   // UNICODE_TO_GBK[12326] := 16#6346;
   // UNICODE_TO_GBK[12327] := 16#C0A6;
   // UNICODE_TO_GBK[12328] := 16#6347;
   // UNICODE_TO_GBK[12329] := 16#92BB;
   // UNICODE_TO_GBK[12330] := 16#6348;
   // UNICODE_TO_GBK[12331] := 16#92BC;
   // UNICODE_TO_GBK[12332] := 16#6349;
   // UNICODE_TO_GBK[12333] := 16#D7BD;
   // UNICODE_TO_GBK[12334] := 16#634A;
   // UNICODE_TO_GBK[12335] := 16#92BD;
   // UNICODE_TO_GBK[12336] := 16#634B;
   // UNICODE_TO_GBK[12337] := 16#DEDB;
   // UNICODE_TO_GBK[12338] := 16#634C;
   // UNICODE_TO_GBK[12339] := 16#B0C6;
   // UNICODE_TO_GBK[12340] := 16#634D;
   // UNICODE_TO_GBK[12341] := 16#BAB4;
   // UNICODE_TO_GBK[12342] := 16#634E;
   // UNICODE_TO_GBK[12343] := 16#C9D3;
   // UNICODE_TO_GBK[12344] := 16#634F;
   // UNICODE_TO_GBK[12345] := 16#C4F3;
   // UNICODE_TO_GBK[12346] := 16#6350;
   // UNICODE_TO_GBK[12347] := 16#BEE8;
   // UNICODE_TO_GBK[12348] := 16#6351;
   // UNICODE_TO_GBK[12349] := 16#92BE;
   // UNICODE_TO_GBK[12350] := 16#6352;
   // UNICODE_TO_GBK[12351] := 16#92BF;
   // UNICODE_TO_GBK[12352] := 16#6353;
   // UNICODE_TO_GBK[12353] := 16#92C0;
   // UNICODE_TO_GBK[12354] := 16#6354;
   // UNICODE_TO_GBK[12355] := 16#92C1;
   // UNICODE_TO_GBK[12356] := 16#6355;
   // UNICODE_TO_GBK[12357] := 16#B2B6;
   // UNICODE_TO_GBK[12358] := 16#6356;
   // UNICODE_TO_GBK[12359] := 16#92C2;
   // UNICODE_TO_GBK[12360] := 16#6357;
   // UNICODE_TO_GBK[12361] := 16#92C3;
   // UNICODE_TO_GBK[12362] := 16#6358;
   // UNICODE_TO_GBK[12363] := 16#92C4;
   // UNICODE_TO_GBK[12364] := 16#6359;
   // UNICODE_TO_GBK[12365] := 16#92C5;
   // UNICODE_TO_GBK[12366] := 16#635A;
   // UNICODE_TO_GBK[12367] := 16#92C6;
   // UNICODE_TO_GBK[12368] := 16#635B;
   // UNICODE_TO_GBK[12369] := 16#92C7;
   // UNICODE_TO_GBK[12370] := 16#635C;
   // UNICODE_TO_GBK[12371] := 16#92C8;
   // UNICODE_TO_GBK[12372] := 16#635D;
   // UNICODE_TO_GBK[12373] := 16#92C9;
   // UNICODE_TO_GBK[12374] := 16#635E;
   // UNICODE_TO_GBK[12375] := 16#C0CC;
   // UNICODE_TO_GBK[12376] := 16#635F;
   // UNICODE_TO_GBK[12377] := 16#CBF0;
   // UNICODE_TO_GBK[12378] := 16#6360;
   // UNICODE_TO_GBK[12379] := 16#92CA;
   // UNICODE_TO_GBK[12380] := 16#6361;
   // UNICODE_TO_GBK[12381] := 16#BCF1;
   // UNICODE_TO_GBK[12382] := 16#6362;
   // UNICODE_TO_GBK[12383] := 16#BBBB;
   // UNICODE_TO_GBK[12384] := 16#6363;
   // UNICODE_TO_GBK[12385] := 16#B5B7;
   // UNICODE_TO_GBK[12386] := 16#6364;
   // UNICODE_TO_GBK[12387] := 16#92CB;
   // UNICODE_TO_GBK[12388] := 16#6365;
   // UNICODE_TO_GBK[12389] := 16#92CC;
   // UNICODE_TO_GBK[12390] := 16#6366;
   // UNICODE_TO_GBK[12391] := 16#92CD;
   // UNICODE_TO_GBK[12392] := 16#6367;
   // UNICODE_TO_GBK[12393] := 16#C5F5;
   // UNICODE_TO_GBK[12394] := 16#6368;
   // UNICODE_TO_GBK[12395] := 16#92CE;
   // UNICODE_TO_GBK[12396] := 16#6369;
   // UNICODE_TO_GBK[12397] := 16#DEE6;
   // UNICODE_TO_GBK[12398] := 16#636A;
   // UNICODE_TO_GBK[12399] := 16#92CF;
   // UNICODE_TO_GBK[12400] := 16#636B;
   // UNICODE_TO_GBK[12401] := 16#92D0;
   // UNICODE_TO_GBK[12402] := 16#636C;
   // UNICODE_TO_GBK[12403] := 16#92D1;
   // UNICODE_TO_GBK[12404] := 16#636D;
   // UNICODE_TO_GBK[12405] := 16#DEE3;
   // UNICODE_TO_GBK[12406] := 16#636E;
   // UNICODE_TO_GBK[12407] := 16#BEDD;
   // UNICODE_TO_GBK[12408] := 16#636F;
   // UNICODE_TO_GBK[12409] := 16#92D2;
   // UNICODE_TO_GBK[12410] := 16#6370;
   // UNICODE_TO_GBK[12411] := 16#92D3;
   // UNICODE_TO_GBK[12412] := 16#6371;
   // UNICODE_TO_GBK[12413] := 16#DEDF;
   // UNICODE_TO_GBK[12414] := 16#6372;
   // UNICODE_TO_GBK[12415] := 16#92D4;
   // UNICODE_TO_GBK[12416] := 16#6373;
   // UNICODE_TO_GBK[12417] := 16#92D5;
   // UNICODE_TO_GBK[12418] := 16#6374;
   // UNICODE_TO_GBK[12419] := 16#92D6;
   // UNICODE_TO_GBK[12420] := 16#6375;
   // UNICODE_TO_GBK[12421] := 16#92D7;
   // UNICODE_TO_GBK[12422] := 16#6376;
   // UNICODE_TO_GBK[12423] := 16#B4B7;
   // UNICODE_TO_GBK[12424] := 16#6377;
   // UNICODE_TO_GBK[12425] := 16#BDDD;
   // UNICODE_TO_GBK[12426] := 16#6378;
   // UNICODE_TO_GBK[12427] := 16#92D8;
   // UNICODE_TO_GBK[12428] := 16#6379;
   // UNICODE_TO_GBK[12429] := 16#92D9;
   // UNICODE_TO_GBK[12430] := 16#637A;
   // UNICODE_TO_GBK[12431] := 16#DEE0;
   // UNICODE_TO_GBK[12432] := 16#637B;
   // UNICODE_TO_GBK[12433] := 16#C4ED;
   // UNICODE_TO_GBK[12434] := 16#637C;
   // UNICODE_TO_GBK[12435] := 16#92DA;
   // UNICODE_TO_GBK[12436] := 16#637D;
   // UNICODE_TO_GBK[12437] := 16#92DB;
   // UNICODE_TO_GBK[12438] := 16#637E;
   // UNICODE_TO_GBK[12439] := 16#92DC;
   // UNICODE_TO_GBK[12440] := 16#637F;
   // UNICODE_TO_GBK[12441] := 16#92DD;
   // UNICODE_TO_GBK[12442] := 16#6380;
   // UNICODE_TO_GBK[12443] := 16#CFC6;
   // UNICODE_TO_GBK[12444] := 16#6381;
   // UNICODE_TO_GBK[12445] := 16#92DE;
   // UNICODE_TO_GBK[12446] := 16#6382;
   // UNICODE_TO_GBK[12447] := 16#B5E0;
   // UNICODE_TO_GBK[12448] := 16#6383;
   // UNICODE_TO_GBK[12449] := 16#92DF;
   // UNICODE_TO_GBK[12450] := 16#6384;
   // UNICODE_TO_GBK[12451] := 16#92E0;
   // UNICODE_TO_GBK[12452] := 16#6385;
   // UNICODE_TO_GBK[12453] := 16#92E1;
   // UNICODE_TO_GBK[12454] := 16#6386;
   // UNICODE_TO_GBK[12455] := 16#92E2;
   // UNICODE_TO_GBK[12456] := 16#6387;
   // UNICODE_TO_GBK[12457] := 16#B6DE;
   // UNICODE_TO_GBK[12458] := 16#6388;
   // UNICODE_TO_GBK[12459] := 16#CADA;
   // UNICODE_TO_GBK[12460] := 16#6389;
   // UNICODE_TO_GBK[12461] := 16#B5F4;
   // UNICODE_TO_GBK[12462] := 16#638A;
   // UNICODE_TO_GBK[12463] := 16#DEE5;
   // UNICODE_TO_GBK[12464] := 16#638B;
   // UNICODE_TO_GBK[12465] := 16#92E3;
   // UNICODE_TO_GBK[12466] := 16#638C;
   // UNICODE_TO_GBK[12467] := 16#D5C6;
   // UNICODE_TO_GBK[12468] := 16#638D;
   // UNICODE_TO_GBK[12469] := 16#92E4;
   // UNICODE_TO_GBK[12470] := 16#638E;
   // UNICODE_TO_GBK[12471] := 16#DEE1;
   // UNICODE_TO_GBK[12472] := 16#638F;
   // UNICODE_TO_GBK[12473] := 16#CCCD;
   // UNICODE_TO_GBK[12474] := 16#6390;
   // UNICODE_TO_GBK[12475] := 16#C6FE;
   // UNICODE_TO_GBK[12476] := 16#6391;
   // UNICODE_TO_GBK[12477] := 16#92E5;
   // UNICODE_TO_GBK[12478] := 16#6392;
   // UNICODE_TO_GBK[12479] := 16#C5C5;
   // UNICODE_TO_GBK[12480] := 16#6393;
   // UNICODE_TO_GBK[12481] := 16#92E6;
   // UNICODE_TO_GBK[12482] := 16#6394;
   // UNICODE_TO_GBK[12483] := 16#92E7;
   // UNICODE_TO_GBK[12484] := 16#6395;
   // UNICODE_TO_GBK[12485] := 16#92E8;
   // UNICODE_TO_GBK[12486] := 16#6396;
   // UNICODE_TO_GBK[12487] := 16#D2B4;
   // UNICODE_TO_GBK[12488] := 16#6397;
   // UNICODE_TO_GBK[12489] := 16#92E9;
   // UNICODE_TO_GBK[12490] := 16#6398;
   // UNICODE_TO_GBK[12491] := 16#BEF2;
   // UNICODE_TO_GBK[12492] := 16#6399;
   // UNICODE_TO_GBK[12493] := 16#92EA;
   // UNICODE_TO_GBK[12494] := 16#639A;
   // UNICODE_TO_GBK[12495] := 16#92EB;
   // UNICODE_TO_GBK[12496] := 16#639B;
   // UNICODE_TO_GBK[12497] := 16#92EC;
   // UNICODE_TO_GBK[12498] := 16#639C;
   // UNICODE_TO_GBK[12499] := 16#92ED;
   // UNICODE_TO_GBK[12500] := 16#639D;
   // UNICODE_TO_GBK[12501] := 16#92EE;
   // UNICODE_TO_GBK[12502] := 16#639E;
   // UNICODE_TO_GBK[12503] := 16#92EF;
   // UNICODE_TO_GBK[12504] := 16#639F;
   // UNICODE_TO_GBK[12505] := 16#92F0;
   // UNICODE_TO_GBK[12506] := 16#63A0;
   // UNICODE_TO_GBK[12507] := 16#C2D3;
   // UNICODE_TO_GBK[12508] := 16#63A1;
   // UNICODE_TO_GBK[12509] := 16#92F1;
   // UNICODE_TO_GBK[12510] := 16#63A2;
   // UNICODE_TO_GBK[12511] := 16#CCBD;
   // UNICODE_TO_GBK[12512] := 16#63A3;
   // UNICODE_TO_GBK[12513] := 16#B3B8;
   // UNICODE_TO_GBK[12514] := 16#63A4;
   // UNICODE_TO_GBK[12515] := 16#92F2;
   // UNICODE_TO_GBK[12516] := 16#63A5;
   // UNICODE_TO_GBK[12517] := 16#BDD3;
   // UNICODE_TO_GBK[12518] := 16#63A6;
   // UNICODE_TO_GBK[12519] := 16#92F3;
   // UNICODE_TO_GBK[12520] := 16#63A7;
   // UNICODE_TO_GBK[12521] := 16#BFD8;
   // UNICODE_TO_GBK[12522] := 16#63A8;
   // UNICODE_TO_GBK[12523] := 16#CDC6;
   // UNICODE_TO_GBK[12524] := 16#63A9;
   // UNICODE_TO_GBK[12525] := 16#D1DA;
   // UNICODE_TO_GBK[12526] := 16#63AA;
   // UNICODE_TO_GBK[12527] := 16#B4EB;
   // UNICODE_TO_GBK[12528] := 16#63AB;
   // UNICODE_TO_GBK[12529] := 16#92F4;
   // UNICODE_TO_GBK[12530] := 16#63AC;
   // UNICODE_TO_GBK[12531] := 16#DEE4;
   // UNICODE_TO_GBK[12532] := 16#63AD;
   // UNICODE_TO_GBK[12533] := 16#DEDD;
   // UNICODE_TO_GBK[12534] := 16#63AE;
   // UNICODE_TO_GBK[12535] := 16#DEE7;
   // UNICODE_TO_GBK[12536] := 16#63AF;
   // UNICODE_TO_GBK[12537] := 16#92F5;
   // UNICODE_TO_GBK[12538] := 16#63B0;
   // UNICODE_TO_GBK[12539] := 16#EAFE;
   // UNICODE_TO_GBK[12540] := 16#63B1;
   // UNICODE_TO_GBK[12541] := 16#92F6;
   // UNICODE_TO_GBK[12542] := 16#63B2;
   // UNICODE_TO_GBK[12543] := 16#92F7;
   // UNICODE_TO_GBK[12544] := 16#63B3;
   // UNICODE_TO_GBK[12545] := 16#C2B0;
   // UNICODE_TO_GBK[12546] := 16#63B4;
   // UNICODE_TO_GBK[12547] := 16#DEE2;
   // UNICODE_TO_GBK[12548] := 16#63B5;
   // UNICODE_TO_GBK[12549] := 16#92F8;
   // UNICODE_TO_GBK[12550] := 16#63B6;
   // UNICODE_TO_GBK[12551] := 16#92F9;
   // UNICODE_TO_GBK[12552] := 16#63B7;
   // UNICODE_TO_GBK[12553] := 16#D6C0;
   // UNICODE_TO_GBK[12554] := 16#63B8;
   // UNICODE_TO_GBK[12555] := 16#B5A7;
   // UNICODE_TO_GBK[12556] := 16#63B9;
   // UNICODE_TO_GBK[12557] := 16#92FA;
   // UNICODE_TO_GBK[12558] := 16#63BA;
   // UNICODE_TO_GBK[12559] := 16#B2F4;
   // UNICODE_TO_GBK[12560] := 16#63BB;
   // UNICODE_TO_GBK[12561] := 16#92FB;
   // UNICODE_TO_GBK[12562] := 16#63BC;
   // UNICODE_TO_GBK[12563] := 16#DEE8;
   // UNICODE_TO_GBK[12564] := 16#63BD;
   // UNICODE_TO_GBK[12565] := 16#92FC;
   // UNICODE_TO_GBK[12566] := 16#63BE;
   // UNICODE_TO_GBK[12567] := 16#DEF2;
   // UNICODE_TO_GBK[12568] := 16#63BF;
   // UNICODE_TO_GBK[12569] := 16#92FD;
   // UNICODE_TO_GBK[12570] := 16#63C0;
   // UNICODE_TO_GBK[12571] := 16#92FE;
   // UNICODE_TO_GBK[12572] := 16#63C1;
   // UNICODE_TO_GBK[12573] := 16#9340;
   // UNICODE_TO_GBK[12574] := 16#63C2;
   // UNICODE_TO_GBK[12575] := 16#9341;
   // UNICODE_TO_GBK[12576] := 16#63C3;
   // UNICODE_TO_GBK[12577] := 16#9342;
   // UNICODE_TO_GBK[12578] := 16#63C4;
   // UNICODE_TO_GBK[12579] := 16#DEED;
   // UNICODE_TO_GBK[12580] := 16#63C5;
   // UNICODE_TO_GBK[12581] := 16#9343;
   // UNICODE_TO_GBK[12582] := 16#63C6;
   // UNICODE_TO_GBK[12583] := 16#DEF1;
   // UNICODE_TO_GBK[12584] := 16#63C7;
   // UNICODE_TO_GBK[12585] := 16#9344;
   // UNICODE_TO_GBK[12586] := 16#63C8;
   // UNICODE_TO_GBK[12587] := 16#9345;
   // UNICODE_TO_GBK[12588] := 16#63C9;
   // UNICODE_TO_GBK[12589] := 16#C8E0;
   // UNICODE_TO_GBK[12590] := 16#63CA;
   // UNICODE_TO_GBK[12591] := 16#9346;
   // UNICODE_TO_GBK[12592] := 16#63CB;
   // UNICODE_TO_GBK[12593] := 16#9347;
   // UNICODE_TO_GBK[12594] := 16#63CC;
   // UNICODE_TO_GBK[12595] := 16#9348;
   // UNICODE_TO_GBK[12596] := 16#63CD;
   // UNICODE_TO_GBK[12597] := 16#D7E1;
   // UNICODE_TO_GBK[12598] := 16#63CE;
   // UNICODE_TO_GBK[12599] := 16#DEEF;
   // UNICODE_TO_GBK[12600] := 16#63CF;
   // UNICODE_TO_GBK[12601] := 16#C3E8;
   // UNICODE_TO_GBK[12602] := 16#63D0;
   // UNICODE_TO_GBK[12603] := 16#CCE1;
   // UNICODE_TO_GBK[12604] := 16#63D1;
   // UNICODE_TO_GBK[12605] := 16#9349;
   // UNICODE_TO_GBK[12606] := 16#63D2;
   // UNICODE_TO_GBK[12607] := 16#B2E5;
   // UNICODE_TO_GBK[12608] := 16#63D3;
   // UNICODE_TO_GBK[12609] := 16#934A;
   // UNICODE_TO_GBK[12610] := 16#63D4;
   // UNICODE_TO_GBK[12611] := 16#934B;
   // UNICODE_TO_GBK[12612] := 16#63D5;
   // UNICODE_TO_GBK[12613] := 16#934C;
   // UNICODE_TO_GBK[12614] := 16#63D6;
   // UNICODE_TO_GBK[12615] := 16#D2BE;
   // UNICODE_TO_GBK[12616] := 16#63D7;
   // UNICODE_TO_GBK[12617] := 16#934D;
   // UNICODE_TO_GBK[12618] := 16#63D8;
   // UNICODE_TO_GBK[12619] := 16#934E;
   // UNICODE_TO_GBK[12620] := 16#63D9;
   // UNICODE_TO_GBK[12621] := 16#934F;
   // UNICODE_TO_GBK[12622] := 16#63DA;
   // UNICODE_TO_GBK[12623] := 16#9350;
   // UNICODE_TO_GBK[12624] := 16#63DB;
   // UNICODE_TO_GBK[12625] := 16#9351;
   // UNICODE_TO_GBK[12626] := 16#63DC;
   // UNICODE_TO_GBK[12627] := 16#9352;
   // UNICODE_TO_GBK[12628] := 16#63DD;
   // UNICODE_TO_GBK[12629] := 16#9353;
   // UNICODE_TO_GBK[12630] := 16#63DE;
   // UNICODE_TO_GBK[12631] := 16#DEEE;
   // UNICODE_TO_GBK[12632] := 16#63DF;
   // UNICODE_TO_GBK[12633] := 16#9354;
   // UNICODE_TO_GBK[12634] := 16#63E0;
   // UNICODE_TO_GBK[12635] := 16#DEEB;
   // UNICODE_TO_GBK[12636] := 16#63E1;
   // UNICODE_TO_GBK[12637] := 16#CED5;
   // UNICODE_TO_GBK[12638] := 16#63E2;
   // UNICODE_TO_GBK[12639] := 16#9355;
   // UNICODE_TO_GBK[12640] := 16#63E3;
   // UNICODE_TO_GBK[12641] := 16#B4A7;
   // UNICODE_TO_GBK[12642] := 16#63E4;
   // UNICODE_TO_GBK[12643] := 16#9356;
   // UNICODE_TO_GBK[12644] := 16#63E5;
   // UNICODE_TO_GBK[12645] := 16#9357;
   // UNICODE_TO_GBK[12646] := 16#63E6;
   // UNICODE_TO_GBK[12647] := 16#9358;
   // UNICODE_TO_GBK[12648] := 16#63E7;
   // UNICODE_TO_GBK[12649] := 16#9359;
   // UNICODE_TO_GBK[12650] := 16#63E8;
   // UNICODE_TO_GBK[12651] := 16#935A;
   // UNICODE_TO_GBK[12652] := 16#63E9;
   // UNICODE_TO_GBK[12653] := 16#BFAB;
   // UNICODE_TO_GBK[12654] := 16#63EA;
   // UNICODE_TO_GBK[12655] := 16#BEBE;
   // UNICODE_TO_GBK[12656] := 16#63EB;
   // UNICODE_TO_GBK[12657] := 16#935B;
   // UNICODE_TO_GBK[12658] := 16#63EC;
   // UNICODE_TO_GBK[12659] := 16#935C;
   // UNICODE_TO_GBK[12660] := 16#63ED;
   // UNICODE_TO_GBK[12661] := 16#BDD2;
   // UNICODE_TO_GBK[12662] := 16#63EE;
   // UNICODE_TO_GBK[12663] := 16#935D;
   // UNICODE_TO_GBK[12664] := 16#63EF;
   // UNICODE_TO_GBK[12665] := 16#935E;
   // UNICODE_TO_GBK[12666] := 16#63F0;
   // UNICODE_TO_GBK[12667] := 16#935F;
   // UNICODE_TO_GBK[12668] := 16#63F1;
   // UNICODE_TO_GBK[12669] := 16#9360;
   // UNICODE_TO_GBK[12670] := 16#63F2;
   // UNICODE_TO_GBK[12671] := 16#DEE9;
   // UNICODE_TO_GBK[12672] := 16#63F3;
   // UNICODE_TO_GBK[12673] := 16#9361;
   // UNICODE_TO_GBK[12674] := 16#63F4;
   // UNICODE_TO_GBK[12675] := 16#D4AE;
   // UNICODE_TO_GBK[12676] := 16#63F5;
   // UNICODE_TO_GBK[12677] := 16#9362;
   // UNICODE_TO_GBK[12678] := 16#63F6;
   // UNICODE_TO_GBK[12679] := 16#DEDE;
   // UNICODE_TO_GBK[12680] := 16#63F7;
   // UNICODE_TO_GBK[12681] := 16#9363;
   // UNICODE_TO_GBK[12682] := 16#63F8;
   // UNICODE_TO_GBK[12683] := 16#DEEA;
   // UNICODE_TO_GBK[12684] := 16#63F9;
   // UNICODE_TO_GBK[12685] := 16#9364;
   // UNICODE_TO_GBK[12686] := 16#63FA;
   // UNICODE_TO_GBK[12687] := 16#9365;
   // UNICODE_TO_GBK[12688] := 16#63FB;
   // UNICODE_TO_GBK[12689] := 16#9366;
   // UNICODE_TO_GBK[12690] := 16#63FC;
   // UNICODE_TO_GBK[12691] := 16#9367;
   // UNICODE_TO_GBK[12692] := 16#63FD;
   // UNICODE_TO_GBK[12693] := 16#C0BF;
   // UNICODE_TO_GBK[12694] := 16#63FE;
   // UNICODE_TO_GBK[12695] := 16#9368;
   // UNICODE_TO_GBK[12696] := 16#63FF;
   // UNICODE_TO_GBK[12697] := 16#DEEC;
   // UNICODE_TO_GBK[12698] := 16#6400;
   // UNICODE_TO_GBK[12699] := 16#B2F3;
   // UNICODE_TO_GBK[12700] := 16#6401;
   // UNICODE_TO_GBK[12701] := 16#B8E9;
   // UNICODE_TO_GBK[12702] := 16#6402;
   // UNICODE_TO_GBK[12703] := 16#C2A7;
   // UNICODE_TO_GBK[12704] := 16#6403;
   // UNICODE_TO_GBK[12705] := 16#9369;
   // UNICODE_TO_GBK[12706] := 16#6404;
   // UNICODE_TO_GBK[12707] := 16#936A;
   // UNICODE_TO_GBK[12708] := 16#6405;
   // UNICODE_TO_GBK[12709] := 16#BDC1;
   // UNICODE_TO_GBK[12710] := 16#6406;
   // UNICODE_TO_GBK[12711] := 16#936B;
   // UNICODE_TO_GBK[12712] := 16#6407;
   // UNICODE_TO_GBK[12713] := 16#936C;
   // UNICODE_TO_GBK[12714] := 16#6408;
   // UNICODE_TO_GBK[12715] := 16#936D;
   // UNICODE_TO_GBK[12716] := 16#6409;
   // UNICODE_TO_GBK[12717] := 16#936E;
   // UNICODE_TO_GBK[12718] := 16#640A;
   // UNICODE_TO_GBK[12719] := 16#936F;
   // UNICODE_TO_GBK[12720] := 16#640B;
   // UNICODE_TO_GBK[12721] := 16#DEF5;
   // UNICODE_TO_GBK[12722] := 16#640C;
   // UNICODE_TO_GBK[12723] := 16#DEF8;
   // UNICODE_TO_GBK[12724] := 16#640D;
   // UNICODE_TO_GBK[12725] := 16#9370;
   // UNICODE_TO_GBK[12726] := 16#640E;
   // UNICODE_TO_GBK[12727] := 16#9371;
   // UNICODE_TO_GBK[12728] := 16#640F;
   // UNICODE_TO_GBK[12729] := 16#B2AB;
   // UNICODE_TO_GBK[12730] := 16#6410;
   // UNICODE_TO_GBK[12731] := 16#B4A4;
   // UNICODE_TO_GBK[12732] := 16#6411;
   // UNICODE_TO_GBK[12733] := 16#9372;
   // UNICODE_TO_GBK[12734] := 16#6412;
   // UNICODE_TO_GBK[12735] := 16#9373;
   // UNICODE_TO_GBK[12736] := 16#6413;
   // UNICODE_TO_GBK[12737] := 16#B4EA;
   // UNICODE_TO_GBK[12738] := 16#6414;
   // UNICODE_TO_GBK[12739] := 16#C9A6;
   // UNICODE_TO_GBK[12740] := 16#6415;
   // UNICODE_TO_GBK[12741] := 16#9374;
   // UNICODE_TO_GBK[12742] := 16#6416;
   // UNICODE_TO_GBK[12743] := 16#9375;
   // UNICODE_TO_GBK[12744] := 16#6417;
   // UNICODE_TO_GBK[12745] := 16#9376;
   // UNICODE_TO_GBK[12746] := 16#6418;
   // UNICODE_TO_GBK[12747] := 16#9377;
   // UNICODE_TO_GBK[12748] := 16#6419;
   // UNICODE_TO_GBK[12749] := 16#9378;
   // UNICODE_TO_GBK[12750] := 16#641A;
   // UNICODE_TO_GBK[12751] := 16#9379;
   // UNICODE_TO_GBK[12752] := 16#641B;
   // UNICODE_TO_GBK[12753] := 16#DEF6;
   // UNICODE_TO_GBK[12754] := 16#641C;
   // UNICODE_TO_GBK[12755] := 16#CBD1;
   // UNICODE_TO_GBK[12756] := 16#641D;
   // UNICODE_TO_GBK[12757] := 16#937A;
   // UNICODE_TO_GBK[12758] := 16#641E;
   // UNICODE_TO_GBK[12759] := 16#B8E3;
   // UNICODE_TO_GBK[12760] := 16#641F;
   // UNICODE_TO_GBK[12761] := 16#937B;
   // UNICODE_TO_GBK[12762] := 16#6420;
   // UNICODE_TO_GBK[12763] := 16#DEF7;
   // UNICODE_TO_GBK[12764] := 16#6421;
   // UNICODE_TO_GBK[12765] := 16#DEFA;
   // UNICODE_TO_GBK[12766] := 16#6422;
   // UNICODE_TO_GBK[12767] := 16#937C;
   // UNICODE_TO_GBK[12768] := 16#6423;
   // UNICODE_TO_GBK[12769] := 16#937D;
   // UNICODE_TO_GBK[12770] := 16#6424;
   // UNICODE_TO_GBK[12771] := 16#937E;
   // UNICODE_TO_GBK[12772] := 16#6425;
   // UNICODE_TO_GBK[12773] := 16#9380;
   // UNICODE_TO_GBK[12774] := 16#6426;
   // UNICODE_TO_GBK[12775] := 16#DEF9;
   // UNICODE_TO_GBK[12776] := 16#6427;
   // UNICODE_TO_GBK[12777] := 16#9381;
   // UNICODE_TO_GBK[12778] := 16#6428;
   // UNICODE_TO_GBK[12779] := 16#9382;
   // UNICODE_TO_GBK[12780] := 16#6429;
   // UNICODE_TO_GBK[12781] := 16#9383;
   // UNICODE_TO_GBK[12782] := 16#642A;
   // UNICODE_TO_GBK[12783] := 16#CCC2;
   // UNICODE_TO_GBK[12784] := 16#642B;
   // UNICODE_TO_GBK[12785] := 16#9384;
   // UNICODE_TO_GBK[12786] := 16#642C;
   // UNICODE_TO_GBK[12787] := 16#B0E1;
   // UNICODE_TO_GBK[12788] := 16#642D;
   // UNICODE_TO_GBK[12789] := 16#B4EE;
   // UNICODE_TO_GBK[12790] := 16#642E;
   // UNICODE_TO_GBK[12791] := 16#9385;
   // UNICODE_TO_GBK[12792] := 16#642F;
   // UNICODE_TO_GBK[12793] := 16#9386;
   // UNICODE_TO_GBK[12794] := 16#6430;
   // UNICODE_TO_GBK[12795] := 16#9387;
   // UNICODE_TO_GBK[12796] := 16#6431;
   // UNICODE_TO_GBK[12797] := 16#9388;
   // UNICODE_TO_GBK[12798] := 16#6432;
   // UNICODE_TO_GBK[12799] := 16#9389;
   // UNICODE_TO_GBK[12800] := 16#6433;
   // UNICODE_TO_GBK[12801] := 16#938A;
   // UNICODE_TO_GBK[12802] := 16#6434;
   // UNICODE_TO_GBK[12803] := 16#E5BA;
   // UNICODE_TO_GBK[12804] := 16#6435;
   // UNICODE_TO_GBK[12805] := 16#938B;
   // UNICODE_TO_GBK[12806] := 16#6436;
   // UNICODE_TO_GBK[12807] := 16#938C;
   // UNICODE_TO_GBK[12808] := 16#6437;
   // UNICODE_TO_GBK[12809] := 16#938D;
   // UNICODE_TO_GBK[12810] := 16#6438;
   // UNICODE_TO_GBK[12811] := 16#938E;
   // UNICODE_TO_GBK[12812] := 16#6439;
   // UNICODE_TO_GBK[12813] := 16#938F;
   // UNICODE_TO_GBK[12814] := 16#643A;
   // UNICODE_TO_GBK[12815] := 16#D0AF;
   // UNICODE_TO_GBK[12816] := 16#643B;
   // UNICODE_TO_GBK[12817] := 16#9390;
   // UNICODE_TO_GBK[12818] := 16#643C;
   // UNICODE_TO_GBK[12819] := 16#9391;
   // UNICODE_TO_GBK[12820] := 16#643D;
   // UNICODE_TO_GBK[12821] := 16#B2EB;
   // UNICODE_TO_GBK[12822] := 16#643E;
   // UNICODE_TO_GBK[12823] := 16#9392;
   // UNICODE_TO_GBK[12824] := 16#643F;
   // UNICODE_TO_GBK[12825] := 16#EBA1;
   // UNICODE_TO_GBK[12826] := 16#6440;
   // UNICODE_TO_GBK[12827] := 16#9393;
   // UNICODE_TO_GBK[12828] := 16#6441;
   // UNICODE_TO_GBK[12829] := 16#DEF4;
   // UNICODE_TO_GBK[12830] := 16#6442;
   // UNICODE_TO_GBK[12831] := 16#9394;
   // UNICODE_TO_GBK[12832] := 16#6443;
   // UNICODE_TO_GBK[12833] := 16#9395;
   // UNICODE_TO_GBK[12834] := 16#6444;
   // UNICODE_TO_GBK[12835] := 16#C9E3;
   // UNICODE_TO_GBK[12836] := 16#6445;
   // UNICODE_TO_GBK[12837] := 16#DEF3;
   // UNICODE_TO_GBK[12838] := 16#6446;
   // UNICODE_TO_GBK[12839] := 16#B0DA;
   // UNICODE_TO_GBK[12840] := 16#6447;
   // UNICODE_TO_GBK[12841] := 16#D2A1;
   // UNICODE_TO_GBK[12842] := 16#6448;
   // UNICODE_TO_GBK[12843] := 16#B1F7;
   // UNICODE_TO_GBK[12844] := 16#6449;
   // UNICODE_TO_GBK[12845] := 16#9396;
   // UNICODE_TO_GBK[12846] := 16#644A;
   // UNICODE_TO_GBK[12847] := 16#CCAF;
   // UNICODE_TO_GBK[12848] := 16#644B;
   // UNICODE_TO_GBK[12849] := 16#9397;
   // UNICODE_TO_GBK[12850] := 16#644C;
   // UNICODE_TO_GBK[12851] := 16#9398;
   // UNICODE_TO_GBK[12852] := 16#644D;
   // UNICODE_TO_GBK[12853] := 16#9399;
   // UNICODE_TO_GBK[12854] := 16#644E;
   // UNICODE_TO_GBK[12855] := 16#939A;
   // UNICODE_TO_GBK[12856] := 16#644F;
   // UNICODE_TO_GBK[12857] := 16#939B;
   // UNICODE_TO_GBK[12858] := 16#6450;
   // UNICODE_TO_GBK[12859] := 16#939C;
   // UNICODE_TO_GBK[12860] := 16#6451;
   // UNICODE_TO_GBK[12861] := 16#939D;
   // UNICODE_TO_GBK[12862] := 16#6452;
   // UNICODE_TO_GBK[12863] := 16#DEF0;
   // UNICODE_TO_GBK[12864] := 16#6453;
   // UNICODE_TO_GBK[12865] := 16#939E;
   // UNICODE_TO_GBK[12866] := 16#6454;
   // UNICODE_TO_GBK[12867] := 16#CBA4;
   // UNICODE_TO_GBK[12868] := 16#6455;
   // UNICODE_TO_GBK[12869] := 16#939F;
   // UNICODE_TO_GBK[12870] := 16#6456;
   // UNICODE_TO_GBK[12871] := 16#93A0;
   // UNICODE_TO_GBK[12872] := 16#6457;
   // UNICODE_TO_GBK[12873] := 16#93A1;
   // UNICODE_TO_GBK[12874] := 16#6458;
   // UNICODE_TO_GBK[12875] := 16#D5AA;
   // UNICODE_TO_GBK[12876] := 16#6459;
   // UNICODE_TO_GBK[12877] := 16#93A2;
   // UNICODE_TO_GBK[12878] := 16#645A;
   // UNICODE_TO_GBK[12879] := 16#93A3;
   // UNICODE_TO_GBK[12880] := 16#645B;
   // UNICODE_TO_GBK[12881] := 16#93A4;
   // UNICODE_TO_GBK[12882] := 16#645C;
   // UNICODE_TO_GBK[12883] := 16#93A5;
   // UNICODE_TO_GBK[12884] := 16#645D;
   // UNICODE_TO_GBK[12885] := 16#93A6;
   // UNICODE_TO_GBK[12886] := 16#645E;
   // UNICODE_TO_GBK[12887] := 16#DEFB;
   // UNICODE_TO_GBK[12888] := 16#645F;
   // UNICODE_TO_GBK[12889] := 16#93A7;
   // UNICODE_TO_GBK[12890] := 16#6460;
   // UNICODE_TO_GBK[12891] := 16#93A8;
   // UNICODE_TO_GBK[12892] := 16#6461;
   // UNICODE_TO_GBK[12893] := 16#93A9;
   // UNICODE_TO_GBK[12894] := 16#6462;
   // UNICODE_TO_GBK[12895] := 16#93AA;
   // UNICODE_TO_GBK[12896] := 16#6463;
   // UNICODE_TO_GBK[12897] := 16#93AB;
   // UNICODE_TO_GBK[12898] := 16#6464;
   // UNICODE_TO_GBK[12899] := 16#93AC;
   // UNICODE_TO_GBK[12900] := 16#6465;
   // UNICODE_TO_GBK[12901] := 16#93AD;
   // UNICODE_TO_GBK[12902] := 16#6466;
   // UNICODE_TO_GBK[12903] := 16#93AE;
   // UNICODE_TO_GBK[12904] := 16#6467;
   // UNICODE_TO_GBK[12905] := 16#B4DD;
   // UNICODE_TO_GBK[12906] := 16#6468;
   // UNICODE_TO_GBK[12907] := 16#93AF;
   // UNICODE_TO_GBK[12908] := 16#6469;
   // UNICODE_TO_GBK[12909] := 16#C4A6;
   // UNICODE_TO_GBK[12910] := 16#646A;
   // UNICODE_TO_GBK[12911] := 16#93B0;
   // UNICODE_TO_GBK[12912] := 16#646B;
   // UNICODE_TO_GBK[12913] := 16#93B1;
   // UNICODE_TO_GBK[12914] := 16#646C;
   // UNICODE_TO_GBK[12915] := 16#93B2;
   // UNICODE_TO_GBK[12916] := 16#646D;
   // UNICODE_TO_GBK[12917] := 16#DEFD;
   // UNICODE_TO_GBK[12918] := 16#646E;
   // UNICODE_TO_GBK[12919] := 16#93B3;
   // UNICODE_TO_GBK[12920] := 16#646F;
   // UNICODE_TO_GBK[12921] := 16#93B4;
   // UNICODE_TO_GBK[12922] := 16#6470;
   // UNICODE_TO_GBK[12923] := 16#93B5;
   // UNICODE_TO_GBK[12924] := 16#6471;
   // UNICODE_TO_GBK[12925] := 16#93B6;
   // UNICODE_TO_GBK[12926] := 16#6472;
   // UNICODE_TO_GBK[12927] := 16#93B7;
   // UNICODE_TO_GBK[12928] := 16#6473;
   // UNICODE_TO_GBK[12929] := 16#93B8;
   // UNICODE_TO_GBK[12930] := 16#6474;
   // UNICODE_TO_GBK[12931] := 16#93B9;
   // UNICODE_TO_GBK[12932] := 16#6475;
   // UNICODE_TO_GBK[12933] := 16#93BA;
   // UNICODE_TO_GBK[12934] := 16#6476;
   // UNICODE_TO_GBK[12935] := 16#93BB;
   // UNICODE_TO_GBK[12936] := 16#6477;
   // UNICODE_TO_GBK[12937] := 16#93BC;
   // UNICODE_TO_GBK[12938] := 16#6478;
   // UNICODE_TO_GBK[12939] := 16#C3FE;
   // UNICODE_TO_GBK[12940] := 16#6479;
   // UNICODE_TO_GBK[12941] := 16#C4A1;
   // UNICODE_TO_GBK[12942] := 16#647A;
   // UNICODE_TO_GBK[12943] := 16#DFA1;
   // UNICODE_TO_GBK[12944] := 16#647B;
   // UNICODE_TO_GBK[12945] := 16#93BD;
   // UNICODE_TO_GBK[12946] := 16#647C;
   // UNICODE_TO_GBK[12947] := 16#93BE;
   // UNICODE_TO_GBK[12948] := 16#647D;
   // UNICODE_TO_GBK[12949] := 16#93BF;
   // UNICODE_TO_GBK[12950] := 16#647E;
   // UNICODE_TO_GBK[12951] := 16#93C0;
   // UNICODE_TO_GBK[12952] := 16#647F;
   // UNICODE_TO_GBK[12953] := 16#93C1;
   // UNICODE_TO_GBK[12954] := 16#6480;
   // UNICODE_TO_GBK[12955] := 16#93C2;
   // UNICODE_TO_GBK[12956] := 16#6481;
   // UNICODE_TO_GBK[12957] := 16#93C3;
   // UNICODE_TO_GBK[12958] := 16#6482;
   // UNICODE_TO_GBK[12959] := 16#C1CC;
   // UNICODE_TO_GBK[12960] := 16#6483;
   // UNICODE_TO_GBK[12961] := 16#93C4;
   // UNICODE_TO_GBK[12962] := 16#6484;
   // UNICODE_TO_GBK[12963] := 16#DEFC;
   // UNICODE_TO_GBK[12964] := 16#6485;
   // UNICODE_TO_GBK[12965] := 16#BEEF;
   // UNICODE_TO_GBK[12966] := 16#6486;
   // UNICODE_TO_GBK[12967] := 16#93C5;
   // UNICODE_TO_GBK[12968] := 16#6487;
   // UNICODE_TO_GBK[12969] := 16#C6B2;
   // UNICODE_TO_GBK[12970] := 16#6488;
   // UNICODE_TO_GBK[12971] := 16#93C6;
   // UNICODE_TO_GBK[12972] := 16#6489;
   // UNICODE_TO_GBK[12973] := 16#93C7;
   // UNICODE_TO_GBK[12974] := 16#648A;
   // UNICODE_TO_GBK[12975] := 16#93C8;
   // UNICODE_TO_GBK[12976] := 16#648B;
   // UNICODE_TO_GBK[12977] := 16#93C9;
   // UNICODE_TO_GBK[12978] := 16#648C;
   // UNICODE_TO_GBK[12979] := 16#93CA;
   // UNICODE_TO_GBK[12980] := 16#648D;
   // UNICODE_TO_GBK[12981] := 16#93CB;
   // UNICODE_TO_GBK[12982] := 16#648E;
   // UNICODE_TO_GBK[12983] := 16#93CC;
   // UNICODE_TO_GBK[12984] := 16#648F;
   // UNICODE_TO_GBK[12985] := 16#93CD;
   // UNICODE_TO_GBK[12986] := 16#6490;
   // UNICODE_TO_GBK[12987] := 16#93CE;
   // UNICODE_TO_GBK[12988] := 16#6491;
   // UNICODE_TO_GBK[12989] := 16#B3C5;
   // UNICODE_TO_GBK[12990] := 16#6492;
   // UNICODE_TO_GBK[12991] := 16#C8F6;
   // UNICODE_TO_GBK[12992] := 16#6493;
   // UNICODE_TO_GBK[12993] := 16#93CF;
   // UNICODE_TO_GBK[12994] := 16#6494;
   // UNICODE_TO_GBK[12995] := 16#93D0;
   // UNICODE_TO_GBK[12996] := 16#6495;
   // UNICODE_TO_GBK[12997] := 16#CBBA;
   // UNICODE_TO_GBK[12998] := 16#6496;
   // UNICODE_TO_GBK[12999] := 16#DEFE;
   // UNICODE_TO_GBK[13000] := 16#6497;
   // UNICODE_TO_GBK[13001] := 16#93D1;
   // UNICODE_TO_GBK[13002] := 16#6498;
   // UNICODE_TO_GBK[13003] := 16#93D2;
   // UNICODE_TO_GBK[13004] := 16#6499;
   // UNICODE_TO_GBK[13005] := 16#DFA4;
   // UNICODE_TO_GBK[13006] := 16#649A;
   // UNICODE_TO_GBK[13007] := 16#93D3;
   // UNICODE_TO_GBK[13008] := 16#649B;
   // UNICODE_TO_GBK[13009] := 16#93D4;
   // UNICODE_TO_GBK[13010] := 16#649C;
   // UNICODE_TO_GBK[13011] := 16#93D5;
   // UNICODE_TO_GBK[13012] := 16#649D;
   // UNICODE_TO_GBK[13013] := 16#93D6;
   // UNICODE_TO_GBK[13014] := 16#649E;
   // UNICODE_TO_GBK[13015] := 16#D7B2;
   // UNICODE_TO_GBK[13016] := 16#649F;
   // UNICODE_TO_GBK[13017] := 16#93D7;
   // UNICODE_TO_GBK[13018] := 16#64A0;
   // UNICODE_TO_GBK[13019] := 16#93D8;
   // UNICODE_TO_GBK[13020] := 16#64A1;
   // UNICODE_TO_GBK[13021] := 16#93D9;
   // UNICODE_TO_GBK[13022] := 16#64A2;
   // UNICODE_TO_GBK[13023] := 16#93DA;
   // UNICODE_TO_GBK[13024] := 16#64A3;
   // UNICODE_TO_GBK[13025] := 16#93DB;
   // UNICODE_TO_GBK[13026] := 16#64A4;
   // UNICODE_TO_GBK[13027] := 16#B3B7;
   // UNICODE_TO_GBK[13028] := 16#64A5;
   // UNICODE_TO_GBK[13029] := 16#93DC;
   // UNICODE_TO_GBK[13030] := 16#64A6;
   // UNICODE_TO_GBK[13031] := 16#93DD;
   // UNICODE_TO_GBK[13032] := 16#64A7;
   // UNICODE_TO_GBK[13033] := 16#93DE;
   // UNICODE_TO_GBK[13034] := 16#64A8;
   // UNICODE_TO_GBK[13035] := 16#93DF;
   // UNICODE_TO_GBK[13036] := 16#64A9;
   // UNICODE_TO_GBK[13037] := 16#C1C3;
   // UNICODE_TO_GBK[13038] := 16#64AA;
   // UNICODE_TO_GBK[13039] := 16#93E0;
   // UNICODE_TO_GBK[13040] := 16#64AB;
   // UNICODE_TO_GBK[13041] := 16#93E1;
   // UNICODE_TO_GBK[13042] := 16#64AC;
   // UNICODE_TO_GBK[13043] := 16#C7CB;
   // UNICODE_TO_GBK[13044] := 16#64AD;
   // UNICODE_TO_GBK[13045] := 16#B2A5;
   // UNICODE_TO_GBK[13046] := 16#64AE;
   // UNICODE_TO_GBK[13047] := 16#B4E9;
   // UNICODE_TO_GBK[13048] := 16#64AF;
   // UNICODE_TO_GBK[13049] := 16#93E2;
   // UNICODE_TO_GBK[13050] := 16#64B0;
   // UNICODE_TO_GBK[13051] := 16#D7AB;
   // UNICODE_TO_GBK[13052] := 16#64B1;
   // UNICODE_TO_GBK[13053] := 16#93E3;
   // UNICODE_TO_GBK[13054] := 16#64B2;
   // UNICODE_TO_GBK[13055] := 16#93E4;
   // UNICODE_TO_GBK[13056] := 16#64B3;
   // UNICODE_TO_GBK[13057] := 16#93E5;
   // UNICODE_TO_GBK[13058] := 16#64B4;
   // UNICODE_TO_GBK[13059] := 16#93E6;
   // UNICODE_TO_GBK[13060] := 16#64B5;
   // UNICODE_TO_GBK[13061] := 16#C4EC;
   // UNICODE_TO_GBK[13062] := 16#64B6;
   // UNICODE_TO_GBK[13063] := 16#93E7;
   // UNICODE_TO_GBK[13064] := 16#64B7;
   // UNICODE_TO_GBK[13065] := 16#DFA2;
   // UNICODE_TO_GBK[13066] := 16#64B8;
   // UNICODE_TO_GBK[13067] := 16#DFA3;
   // UNICODE_TO_GBK[13068] := 16#64B9;
   // UNICODE_TO_GBK[13069] := 16#93E8;
   // UNICODE_TO_GBK[13070] := 16#64BA;
   // UNICODE_TO_GBK[13071] := 16#DFA5;
   // UNICODE_TO_GBK[13072] := 16#64BB;
   // UNICODE_TO_GBK[13073] := 16#93E9;
   // UNICODE_TO_GBK[13074] := 16#64BC;
   // UNICODE_TO_GBK[13075] := 16#BAB3;
   // UNICODE_TO_GBK[13076] := 16#64BD;
   // UNICODE_TO_GBK[13077] := 16#93EA;
   // UNICODE_TO_GBK[13078] := 16#64BE;
   // UNICODE_TO_GBK[13079] := 16#93EB;
   // UNICODE_TO_GBK[13080] := 16#64BF;
   // UNICODE_TO_GBK[13081] := 16#93EC;
   // UNICODE_TO_GBK[13082] := 16#64C0;
   // UNICODE_TO_GBK[13083] := 16#DFA6;
   // UNICODE_TO_GBK[13084] := 16#64C1;
   // UNICODE_TO_GBK[13085] := 16#93ED;
   // UNICODE_TO_GBK[13086] := 16#64C2;
   // UNICODE_TO_GBK[13087] := 16#C0DE;
   // UNICODE_TO_GBK[13088] := 16#64C3;
   // UNICODE_TO_GBK[13089] := 16#93EE;
   // UNICODE_TO_GBK[13090] := 16#64C4;
   // UNICODE_TO_GBK[13091] := 16#93EF;
   // UNICODE_TO_GBK[13092] := 16#64C5;
   // UNICODE_TO_GBK[13093] := 16#C9C3;
   // UNICODE_TO_GBK[13094] := 16#64C6;
   // UNICODE_TO_GBK[13095] := 16#93F0;
   // UNICODE_TO_GBK[13096] := 16#64C7;
   // UNICODE_TO_GBK[13097] := 16#93F1;
   // UNICODE_TO_GBK[13098] := 16#64C8;
   // UNICODE_TO_GBK[13099] := 16#93F2;
   // UNICODE_TO_GBK[13100] := 16#64C9;
   // UNICODE_TO_GBK[13101] := 16#93F3;
   // UNICODE_TO_GBK[13102] := 16#64CA;
   // UNICODE_TO_GBK[13103] := 16#93F4;
   // UNICODE_TO_GBK[13104] := 16#64CB;
   // UNICODE_TO_GBK[13105] := 16#93F5;
   // UNICODE_TO_GBK[13106] := 16#64CC;
   // UNICODE_TO_GBK[13107] := 16#93F6;
   // UNICODE_TO_GBK[13108] := 16#64CD;
   // UNICODE_TO_GBK[13109] := 16#B2D9;
   // UNICODE_TO_GBK[13110] := 16#64CE;
   // UNICODE_TO_GBK[13111] := 16#C7E6;
   // UNICODE_TO_GBK[13112] := 16#64CF;
   // UNICODE_TO_GBK[13113] := 16#93F7;
   // UNICODE_TO_GBK[13114] := 16#64D0;
   // UNICODE_TO_GBK[13115] := 16#DFA7;
   // UNICODE_TO_GBK[13116] := 16#64D1;
   // UNICODE_TO_GBK[13117] := 16#93F8;
   // UNICODE_TO_GBK[13118] := 16#64D2;
   // UNICODE_TO_GBK[13119] := 16#C7DC;
   // UNICODE_TO_GBK[13120] := 16#64D3;
   // UNICODE_TO_GBK[13121] := 16#93F9;
   // UNICODE_TO_GBK[13122] := 16#64D4;
   // UNICODE_TO_GBK[13123] := 16#93FA;
   // UNICODE_TO_GBK[13124] := 16#64D5;
   // UNICODE_TO_GBK[13125] := 16#93FB;
   // UNICODE_TO_GBK[13126] := 16#64D6;
   // UNICODE_TO_GBK[13127] := 16#93FC;
   // UNICODE_TO_GBK[13128] := 16#64D7;
   // UNICODE_TO_GBK[13129] := 16#DFA8;
   // UNICODE_TO_GBK[13130] := 16#64D8;
   // UNICODE_TO_GBK[13131] := 16#EBA2;
   // UNICODE_TO_GBK[13132] := 16#64D9;
   // UNICODE_TO_GBK[13133] := 16#93FD;
   // UNICODE_TO_GBK[13134] := 16#64DA;
   // UNICODE_TO_GBK[13135] := 16#93FE;
   // UNICODE_TO_GBK[13136] := 16#64DB;
   // UNICODE_TO_GBK[13137] := 16#9440;
   // UNICODE_TO_GBK[13138] := 16#64DC;
   // UNICODE_TO_GBK[13139] := 16#9441;
   // UNICODE_TO_GBK[13140] := 16#64DD;
   // UNICODE_TO_GBK[13141] := 16#9442;
   // UNICODE_TO_GBK[13142] := 16#64DE;
   // UNICODE_TO_GBK[13143] := 16#CBD3;
   // UNICODE_TO_GBK[13144] := 16#64DF;
   // UNICODE_TO_GBK[13145] := 16#9443;
   // UNICODE_TO_GBK[13146] := 16#64E0;
   // UNICODE_TO_GBK[13147] := 16#9444;
   // UNICODE_TO_GBK[13148] := 16#64E1;
   // UNICODE_TO_GBK[13149] := 16#9445;
   // UNICODE_TO_GBK[13150] := 16#64E2;
   // UNICODE_TO_GBK[13151] := 16#DFAA;
   // UNICODE_TO_GBK[13152] := 16#64E3;
   // UNICODE_TO_GBK[13153] := 16#9446;
   // UNICODE_TO_GBK[13154] := 16#64E4;
   // UNICODE_TO_GBK[13155] := 16#DFA9;
   // UNICODE_TO_GBK[13156] := 16#64E5;
   // UNICODE_TO_GBK[13157] := 16#9447;
   // UNICODE_TO_GBK[13158] := 16#64E6;
   // UNICODE_TO_GBK[13159] := 16#B2C1;
   // UNICODE_TO_GBK[13160] := 16#64E7;
   // UNICODE_TO_GBK[13161] := 16#9448;
   // UNICODE_TO_GBK[13162] := 16#64E8;
   // UNICODE_TO_GBK[13163] := 16#9449;
   // UNICODE_TO_GBK[13164] := 16#64E9;
   // UNICODE_TO_GBK[13165] := 16#944A;
   // UNICODE_TO_GBK[13166] := 16#64EA;
   // UNICODE_TO_GBK[13167] := 16#944B;
   // UNICODE_TO_GBK[13168] := 16#64EB;
   // UNICODE_TO_GBK[13169] := 16#944C;
   // UNICODE_TO_GBK[13170] := 16#64EC;
   // UNICODE_TO_GBK[13171] := 16#944D;
   // UNICODE_TO_GBK[13172] := 16#64ED;
   // UNICODE_TO_GBK[13173] := 16#944E;
   // UNICODE_TO_GBK[13174] := 16#64EE;
   // UNICODE_TO_GBK[13175] := 16#944F;
   // UNICODE_TO_GBK[13176] := 16#64EF;
   // UNICODE_TO_GBK[13177] := 16#9450;
   // UNICODE_TO_GBK[13178] := 16#64F0;
   // UNICODE_TO_GBK[13179] := 16#9451;
   // UNICODE_TO_GBK[13180] := 16#64F1;
   // UNICODE_TO_GBK[13181] := 16#9452;
   // UNICODE_TO_GBK[13182] := 16#64F2;
   // UNICODE_TO_GBK[13183] := 16#9453;
   // UNICODE_TO_GBK[13184] := 16#64F3;
   // UNICODE_TO_GBK[13185] := 16#9454;
   // UNICODE_TO_GBK[13186] := 16#64F4;
   // UNICODE_TO_GBK[13187] := 16#9455;
   // UNICODE_TO_GBK[13188] := 16#64F5;
   // UNICODE_TO_GBK[13189] := 16#9456;
   // UNICODE_TO_GBK[13190] := 16#64F6;
   // UNICODE_TO_GBK[13191] := 16#9457;
   // UNICODE_TO_GBK[13192] := 16#64F7;
   // UNICODE_TO_GBK[13193] := 16#9458;
   // UNICODE_TO_GBK[13194] := 16#64F8;
   // UNICODE_TO_GBK[13195] := 16#9459;
   // UNICODE_TO_GBK[13196] := 16#64F9;
   // UNICODE_TO_GBK[13197] := 16#945A;
   // UNICODE_TO_GBK[13198] := 16#64FA;
   // UNICODE_TO_GBK[13199] := 16#945B;
   // UNICODE_TO_GBK[13200] := 16#64FB;
   // UNICODE_TO_GBK[13201] := 16#945C;
   // UNICODE_TO_GBK[13202] := 16#64FC;
   // UNICODE_TO_GBK[13203] := 16#945D;
   // UNICODE_TO_GBK[13204] := 16#64FD;
   // UNICODE_TO_GBK[13205] := 16#945E;
   // UNICODE_TO_GBK[13206] := 16#64FE;
   // UNICODE_TO_GBK[13207] := 16#945F;
   // UNICODE_TO_GBK[13208] := 16#64FF;
   // UNICODE_TO_GBK[13209] := 16#9460;
   // UNICODE_TO_GBK[13210] := 16#6500;
   // UNICODE_TO_GBK[13211] := 16#C5CA;
   // UNICODE_TO_GBK[13212] := 16#6501;
   // UNICODE_TO_GBK[13213] := 16#9461;
   // UNICODE_TO_GBK[13214] := 16#6502;
   // UNICODE_TO_GBK[13215] := 16#9462;
   // UNICODE_TO_GBK[13216] := 16#6503;
   // UNICODE_TO_GBK[13217] := 16#9463;
   // UNICODE_TO_GBK[13218] := 16#6504;
   // UNICODE_TO_GBK[13219] := 16#9464;
   // UNICODE_TO_GBK[13220] := 16#6505;
   // UNICODE_TO_GBK[13221] := 16#9465;
   // UNICODE_TO_GBK[13222] := 16#6506;
   // UNICODE_TO_GBK[13223] := 16#9466;
   // UNICODE_TO_GBK[13224] := 16#6507;
   // UNICODE_TO_GBK[13225] := 16#9467;
   // UNICODE_TO_GBK[13226] := 16#6508;
   // UNICODE_TO_GBK[13227] := 16#9468;
   // UNICODE_TO_GBK[13228] := 16#6509;
   // UNICODE_TO_GBK[13229] := 16#DFAB;
   // UNICODE_TO_GBK[13230] := 16#650A;
   // UNICODE_TO_GBK[13231] := 16#9469;
   // UNICODE_TO_GBK[13232] := 16#650B;
   // UNICODE_TO_GBK[13233] := 16#946A;
   // UNICODE_TO_GBK[13234] := 16#650C;
   // UNICODE_TO_GBK[13235] := 16#946B;
   // UNICODE_TO_GBK[13236] := 16#650D;
   // UNICODE_TO_GBK[13237] := 16#946C;
   // UNICODE_TO_GBK[13238] := 16#650E;
   // UNICODE_TO_GBK[13239] := 16#946D;
   // UNICODE_TO_GBK[13240] := 16#650F;
   // UNICODE_TO_GBK[13241] := 16#946E;
   // UNICODE_TO_GBK[13242] := 16#6510;
   // UNICODE_TO_GBK[13243] := 16#946F;
   // UNICODE_TO_GBK[13244] := 16#6511;
   // UNICODE_TO_GBK[13245] := 16#9470;
   // UNICODE_TO_GBK[13246] := 16#6512;
   // UNICODE_TO_GBK[13247] := 16#D4DC;
   // UNICODE_TO_GBK[13248] := 16#6513;
   // UNICODE_TO_GBK[13249] := 16#9471;
   // UNICODE_TO_GBK[13250] := 16#6514;
   // UNICODE_TO_GBK[13251] := 16#9472;
   // UNICODE_TO_GBK[13252] := 16#6515;
   // UNICODE_TO_GBK[13253] := 16#9473;
   // UNICODE_TO_GBK[13254] := 16#6516;
   // UNICODE_TO_GBK[13255] := 16#9474;
   // UNICODE_TO_GBK[13256] := 16#6517;
   // UNICODE_TO_GBK[13257] := 16#9475;
   // UNICODE_TO_GBK[13258] := 16#6518;
   // UNICODE_TO_GBK[13259] := 16#C8C1;
   // UNICODE_TO_GBK[13260] := 16#6519;
   // UNICODE_TO_GBK[13261] := 16#9476;
   // UNICODE_TO_GBK[13262] := 16#651A;
   // UNICODE_TO_GBK[13263] := 16#9477;
   // UNICODE_TO_GBK[13264] := 16#651B;
   // UNICODE_TO_GBK[13265] := 16#9478;
   // UNICODE_TO_GBK[13266] := 16#651C;
   // UNICODE_TO_GBK[13267] := 16#9479;
   // UNICODE_TO_GBK[13268] := 16#651D;
   // UNICODE_TO_GBK[13269] := 16#947A;
   // UNICODE_TO_GBK[13270] := 16#651E;
   // UNICODE_TO_GBK[13271] := 16#947B;
   // UNICODE_TO_GBK[13272] := 16#651F;
   // UNICODE_TO_GBK[13273] := 16#947C;
   // UNICODE_TO_GBK[13274] := 16#6520;
   // UNICODE_TO_GBK[13275] := 16#947D;
   // UNICODE_TO_GBK[13276] := 16#6521;
   // UNICODE_TO_GBK[13277] := 16#947E;
   // UNICODE_TO_GBK[13278] := 16#6522;
   // UNICODE_TO_GBK[13279] := 16#9480;
   // UNICODE_TO_GBK[13280] := 16#6523;
   // UNICODE_TO_GBK[13281] := 16#9481;
   // UNICODE_TO_GBK[13282] := 16#6524;
   // UNICODE_TO_GBK[13283] := 16#9482;
   // UNICODE_TO_GBK[13284] := 16#6525;
   // UNICODE_TO_GBK[13285] := 16#DFAC;
   // UNICODE_TO_GBK[13286] := 16#6526;
   // UNICODE_TO_GBK[13287] := 16#9483;
   // UNICODE_TO_GBK[13288] := 16#6527;
   // UNICODE_TO_GBK[13289] := 16#9484;
   // UNICODE_TO_GBK[13290] := 16#6528;
   // UNICODE_TO_GBK[13291] := 16#9485;
   // UNICODE_TO_GBK[13292] := 16#6529;
   // UNICODE_TO_GBK[13293] := 16#9486;
   // UNICODE_TO_GBK[13294] := 16#652A;
   // UNICODE_TO_GBK[13295] := 16#9487;
   // UNICODE_TO_GBK[13296] := 16#652B;
   // UNICODE_TO_GBK[13297] := 16#BEF0;
   // UNICODE_TO_GBK[13298] := 16#652C;
   // UNICODE_TO_GBK[13299] := 16#9488;
   // UNICODE_TO_GBK[13300] := 16#652D;
   // UNICODE_TO_GBK[13301] := 16#9489;
   // UNICODE_TO_GBK[13302] := 16#652E;
   // UNICODE_TO_GBK[13303] := 16#DFAD;
   // UNICODE_TO_GBK[13304] := 16#652F;
   // UNICODE_TO_GBK[13305] := 16#D6A7;
   // UNICODE_TO_GBK[13306] := 16#6530;
   // UNICODE_TO_GBK[13307] := 16#948A;
   // UNICODE_TO_GBK[13308] := 16#6531;
   // UNICODE_TO_GBK[13309] := 16#948B;
   // UNICODE_TO_GBK[13310] := 16#6532;
   // UNICODE_TO_GBK[13311] := 16#948C;
   // UNICODE_TO_GBK[13312] := 16#6533;
   // UNICODE_TO_GBK[13313] := 16#948D;
   // UNICODE_TO_GBK[13314] := 16#6534;
   // UNICODE_TO_GBK[13315] := 16#EAB7;
   // UNICODE_TO_GBK[13316] := 16#6535;
   // UNICODE_TO_GBK[13317] := 16#EBB6;
   // UNICODE_TO_GBK[13318] := 16#6536;
   // UNICODE_TO_GBK[13319] := 16#CAD5;
   // UNICODE_TO_GBK[13320] := 16#6537;
   // UNICODE_TO_GBK[13321] := 16#948E;
   // UNICODE_TO_GBK[13322] := 16#6538;
   // UNICODE_TO_GBK[13323] := 16#D8FC;
   // UNICODE_TO_GBK[13324] := 16#6539;
   // UNICODE_TO_GBK[13325] := 16#B8C4;
   // UNICODE_TO_GBK[13326] := 16#653A;
   // UNICODE_TO_GBK[13327] := 16#948F;
   // UNICODE_TO_GBK[13328] := 16#653B;
   // UNICODE_TO_GBK[13329] := 16#B9A5;
   // UNICODE_TO_GBK[13330] := 16#653C;
   // UNICODE_TO_GBK[13331] := 16#9490;
   // UNICODE_TO_GBK[13332] := 16#653D;
   // UNICODE_TO_GBK[13333] := 16#9491;
   // UNICODE_TO_GBK[13334] := 16#653E;
   // UNICODE_TO_GBK[13335] := 16#B7C5;
   // UNICODE_TO_GBK[13336] := 16#653F;
   // UNICODE_TO_GBK[13337] := 16#D5FE;
   // UNICODE_TO_GBK[13338] := 16#6540;
   // UNICODE_TO_GBK[13339] := 16#9492;
   // UNICODE_TO_GBK[13340] := 16#6541;
   // UNICODE_TO_GBK[13341] := 16#9493;
   // UNICODE_TO_GBK[13342] := 16#6542;
   // UNICODE_TO_GBK[13343] := 16#9494;
   // UNICODE_TO_GBK[13344] := 16#6543;
   // UNICODE_TO_GBK[13345] := 16#9495;
   // UNICODE_TO_GBK[13346] := 16#6544;
   // UNICODE_TO_GBK[13347] := 16#9496;
   // UNICODE_TO_GBK[13348] := 16#6545;
   // UNICODE_TO_GBK[13349] := 16#B9CA;
   // UNICODE_TO_GBK[13350] := 16#6546;
   // UNICODE_TO_GBK[13351] := 16#9497;
   // UNICODE_TO_GBK[13352] := 16#6547;
   // UNICODE_TO_GBK[13353] := 16#9498;
   // UNICODE_TO_GBK[13354] := 16#6548;
   // UNICODE_TO_GBK[13355] := 16#D0A7;
   // UNICODE_TO_GBK[13356] := 16#6549;
   // UNICODE_TO_GBK[13357] := 16#F4CD;
   // UNICODE_TO_GBK[13358] := 16#654A;
   // UNICODE_TO_GBK[13359] := 16#9499;
   // UNICODE_TO_GBK[13360] := 16#654B;
   // UNICODE_TO_GBK[13361] := 16#949A;
   // UNICODE_TO_GBK[13362] := 16#654C;
   // UNICODE_TO_GBK[13363] := 16#B5D0;
   // UNICODE_TO_GBK[13364] := 16#654D;
   // UNICODE_TO_GBK[13365] := 16#949B;
   // UNICODE_TO_GBK[13366] := 16#654E;
   // UNICODE_TO_GBK[13367] := 16#949C;
   // UNICODE_TO_GBK[13368] := 16#654F;
   // UNICODE_TO_GBK[13369] := 16#C3F4;
   // UNICODE_TO_GBK[13370] := 16#6550;
   // UNICODE_TO_GBK[13371] := 16#949D;
   // UNICODE_TO_GBK[13372] := 16#6551;
   // UNICODE_TO_GBK[13373] := 16#BEC8;
   // UNICODE_TO_GBK[13374] := 16#6552;
   // UNICODE_TO_GBK[13375] := 16#949E;
   // UNICODE_TO_GBK[13376] := 16#6553;
   // UNICODE_TO_GBK[13377] := 16#949F;
   // UNICODE_TO_GBK[13378] := 16#6554;
   // UNICODE_TO_GBK[13379] := 16#94A0;
   // UNICODE_TO_GBK[13380] := 16#6555;
   // UNICODE_TO_GBK[13381] := 16#EBB7;
   // UNICODE_TO_GBK[13382] := 16#6556;
   // UNICODE_TO_GBK[13383] := 16#B0BD;
   // UNICODE_TO_GBK[13384] := 16#6557;
   // UNICODE_TO_GBK[13385] := 16#94A1;
   // UNICODE_TO_GBK[13386] := 16#6558;
   // UNICODE_TO_GBK[13387] := 16#94A2;
   // UNICODE_TO_GBK[13388] := 16#6559;
   // UNICODE_TO_GBK[13389] := 16#BDCC;
   // UNICODE_TO_GBK[13390] := 16#655A;
   // UNICODE_TO_GBK[13391] := 16#94A3;
   // UNICODE_TO_GBK[13392] := 16#655B;
   // UNICODE_TO_GBK[13393] := 16#C1B2;
   // UNICODE_TO_GBK[13394] := 16#655C;
   // UNICODE_TO_GBK[13395] := 16#94A4;
   // UNICODE_TO_GBK[13396] := 16#655D;
   // UNICODE_TO_GBK[13397] := 16#B1D6;
   // UNICODE_TO_GBK[13398] := 16#655E;
   // UNICODE_TO_GBK[13399] := 16#B3A8;
   // UNICODE_TO_GBK[13400] := 16#655F;
   // UNICODE_TO_GBK[13401] := 16#94A5;
   // UNICODE_TO_GBK[13402] := 16#6560;
   // UNICODE_TO_GBK[13403] := 16#94A6;
   // UNICODE_TO_GBK[13404] := 16#6561;
   // UNICODE_TO_GBK[13405] := 16#94A7;
   // UNICODE_TO_GBK[13406] := 16#6562;
   // UNICODE_TO_GBK[13407] := 16#B8D2;
   // UNICODE_TO_GBK[13408] := 16#6563;
   // UNICODE_TO_GBK[13409] := 16#C9A2;
   // UNICODE_TO_GBK[13410] := 16#6564;
   // UNICODE_TO_GBK[13411] := 16#94A8;
   // UNICODE_TO_GBK[13412] := 16#6565;
   // UNICODE_TO_GBK[13413] := 16#94A9;
   // UNICODE_TO_GBK[13414] := 16#6566;
   // UNICODE_TO_GBK[13415] := 16#B6D8;
   // UNICODE_TO_GBK[13416] := 16#6567;
   // UNICODE_TO_GBK[13417] := 16#94AA;
   // UNICODE_TO_GBK[13418] := 16#6568;
   // UNICODE_TO_GBK[13419] := 16#94AB;
   // UNICODE_TO_GBK[13420] := 16#6569;
   // UNICODE_TO_GBK[13421] := 16#94AC;
   // UNICODE_TO_GBK[13422] := 16#656A;
   // UNICODE_TO_GBK[13423] := 16#94AD;
   // UNICODE_TO_GBK[13424] := 16#656B;
   // UNICODE_TO_GBK[13425] := 16#EBB8;
   // UNICODE_TO_GBK[13426] := 16#656C;
   // UNICODE_TO_GBK[13427] := 16#BEB4;
   // UNICODE_TO_GBK[13428] := 16#656D;
   // UNICODE_TO_GBK[13429] := 16#94AE;
   // UNICODE_TO_GBK[13430] := 16#656E;
   // UNICODE_TO_GBK[13431] := 16#94AF;
   // UNICODE_TO_GBK[13432] := 16#656F;
   // UNICODE_TO_GBK[13433] := 16#94B0;
   // UNICODE_TO_GBK[13434] := 16#6570;
   // UNICODE_TO_GBK[13435] := 16#CAFD;
   // UNICODE_TO_GBK[13436] := 16#6571;
   // UNICODE_TO_GBK[13437] := 16#94B1;
   // UNICODE_TO_GBK[13438] := 16#6572;
   // UNICODE_TO_GBK[13439] := 16#C7C3;
   // UNICODE_TO_GBK[13440] := 16#6573;
   // UNICODE_TO_GBK[13441] := 16#94B2;
   // UNICODE_TO_GBK[13442] := 16#6574;
   // UNICODE_TO_GBK[13443] := 16#D5FB;
   // UNICODE_TO_GBK[13444] := 16#6575;
   // UNICODE_TO_GBK[13445] := 16#94B3;
   // UNICODE_TO_GBK[13446] := 16#6576;
   // UNICODE_TO_GBK[13447] := 16#94B4;
   // UNICODE_TO_GBK[13448] := 16#6577;
   // UNICODE_TO_GBK[13449] := 16#B7F3;
   // UNICODE_TO_GBK[13450] := 16#6578;
   // UNICODE_TO_GBK[13451] := 16#94B5;
   // UNICODE_TO_GBK[13452] := 16#6579;
   // UNICODE_TO_GBK[13453] := 16#94B6;
   // UNICODE_TO_GBK[13454] := 16#657A;
   // UNICODE_TO_GBK[13455] := 16#94B7;
   // UNICODE_TO_GBK[13456] := 16#657B;
   // UNICODE_TO_GBK[13457] := 16#94B8;
   // UNICODE_TO_GBK[13458] := 16#657C;
   // UNICODE_TO_GBK[13459] := 16#94B9;
   // UNICODE_TO_GBK[13460] := 16#657D;
   // UNICODE_TO_GBK[13461] := 16#94BA;
   // UNICODE_TO_GBK[13462] := 16#657E;
   // UNICODE_TO_GBK[13463] := 16#94BB;
   // UNICODE_TO_GBK[13464] := 16#657F;
   // UNICODE_TO_GBK[13465] := 16#94BC;
   // UNICODE_TO_GBK[13466] := 16#6580;
   // UNICODE_TO_GBK[13467] := 16#94BD;
   // UNICODE_TO_GBK[13468] := 16#6581;
   // UNICODE_TO_GBK[13469] := 16#94BE;
   // UNICODE_TO_GBK[13470] := 16#6582;
   // UNICODE_TO_GBK[13471] := 16#94BF;
   // UNICODE_TO_GBK[13472] := 16#6583;
   // UNICODE_TO_GBK[13473] := 16#94C0;
   // UNICODE_TO_GBK[13474] := 16#6584;
   // UNICODE_TO_GBK[13475] := 16#94C1;
   // UNICODE_TO_GBK[13476] := 16#6585;
   // UNICODE_TO_GBK[13477] := 16#94C2;
   // UNICODE_TO_GBK[13478] := 16#6586;
   // UNICODE_TO_GBK[13479] := 16#94C3;
   // UNICODE_TO_GBK[13480] := 16#6587;
   // UNICODE_TO_GBK[13481] := 16#CEC4;
   // UNICODE_TO_GBK[13482] := 16#6588;
   // UNICODE_TO_GBK[13483] := 16#94C4;
   // UNICODE_TO_GBK[13484] := 16#6589;
   // UNICODE_TO_GBK[13485] := 16#94C5;
   // UNICODE_TO_GBK[13486] := 16#658A;
   // UNICODE_TO_GBK[13487] := 16#94C6;
   // UNICODE_TO_GBK[13488] := 16#658B;
   // UNICODE_TO_GBK[13489] := 16#D5AB;
   // UNICODE_TO_GBK[13490] := 16#658C;
   // UNICODE_TO_GBK[13491] := 16#B1F3;
   // UNICODE_TO_GBK[13492] := 16#658D;
   // UNICODE_TO_GBK[13493] := 16#94C7;
   // UNICODE_TO_GBK[13494] := 16#658E;
   // UNICODE_TO_GBK[13495] := 16#94C8;
   // UNICODE_TO_GBK[13496] := 16#658F;
   // UNICODE_TO_GBK[13497] := 16#94C9;
   // UNICODE_TO_GBK[13498] := 16#6590;
   // UNICODE_TO_GBK[13499] := 16#ECB3;
   // UNICODE_TO_GBK[13500] := 16#6591;
   // UNICODE_TO_GBK[13501] := 16#B0DF;
   // UNICODE_TO_GBK[13502] := 16#6592;
   // UNICODE_TO_GBK[13503] := 16#94CA;
   // UNICODE_TO_GBK[13504] := 16#6593;
   // UNICODE_TO_GBK[13505] := 16#ECB5;
   // UNICODE_TO_GBK[13506] := 16#6594;
   // UNICODE_TO_GBK[13507] := 16#94CB;
   // UNICODE_TO_GBK[13508] := 16#6595;
   // UNICODE_TO_GBK[13509] := 16#94CC;
   // UNICODE_TO_GBK[13510] := 16#6596;
   // UNICODE_TO_GBK[13511] := 16#94CD;
   // UNICODE_TO_GBK[13512] := 16#6597;
   // UNICODE_TO_GBK[13513] := 16#B6B7;
   // UNICODE_TO_GBK[13514] := 16#6598;
   // UNICODE_TO_GBK[13515] := 16#94CE;
   // UNICODE_TO_GBK[13516] := 16#6599;
   // UNICODE_TO_GBK[13517] := 16#C1CF;
   // UNICODE_TO_GBK[13518] := 16#659A;
   // UNICODE_TO_GBK[13519] := 16#94CF;
   // UNICODE_TO_GBK[13520] := 16#659B;
   // UNICODE_TO_GBK[13521] := 16#F5FA;
   // UNICODE_TO_GBK[13522] := 16#659C;
   // UNICODE_TO_GBK[13523] := 16#D0B1;
   // UNICODE_TO_GBK[13524] := 16#659D;
   // UNICODE_TO_GBK[13525] := 16#94D0;
   // UNICODE_TO_GBK[13526] := 16#659E;
   // UNICODE_TO_GBK[13527] := 16#94D1;
   // UNICODE_TO_GBK[13528] := 16#659F;
   // UNICODE_TO_GBK[13529] := 16#D5E5;
   // UNICODE_TO_GBK[13530] := 16#65A0;
   // UNICODE_TO_GBK[13531] := 16#94D2;
   // UNICODE_TO_GBK[13532] := 16#65A1;
   // UNICODE_TO_GBK[13533] := 16#CED3;
   // UNICODE_TO_GBK[13534] := 16#65A2;
   // UNICODE_TO_GBK[13535] := 16#94D3;
   // UNICODE_TO_GBK[13536] := 16#65A3;
   // UNICODE_TO_GBK[13537] := 16#94D4;
   // UNICODE_TO_GBK[13538] := 16#65A4;
   // UNICODE_TO_GBK[13539] := 16#BDEF;
   // UNICODE_TO_GBK[13540] := 16#65A5;
   // UNICODE_TO_GBK[13541] := 16#B3E2;
   // UNICODE_TO_GBK[13542] := 16#65A6;
   // UNICODE_TO_GBK[13543] := 16#94D5;
   // UNICODE_TO_GBK[13544] := 16#65A7;
   // UNICODE_TO_GBK[13545] := 16#B8AB;
   // UNICODE_TO_GBK[13546] := 16#65A8;
   // UNICODE_TO_GBK[13547] := 16#94D6;
   // UNICODE_TO_GBK[13548] := 16#65A9;
   // UNICODE_TO_GBK[13549] := 16#D5B6;
   // UNICODE_TO_GBK[13550] := 16#65AA;
   // UNICODE_TO_GBK[13551] := 16#94D7;
   // UNICODE_TO_GBK[13552] := 16#65AB;
   // UNICODE_TO_GBK[13553] := 16#EDBD;
   // UNICODE_TO_GBK[13554] := 16#65AC;
   // UNICODE_TO_GBK[13555] := 16#94D8;
   // UNICODE_TO_GBK[13556] := 16#65AD;
   // UNICODE_TO_GBK[13557] := 16#B6CF;
   // UNICODE_TO_GBK[13558] := 16#65AE;
   // UNICODE_TO_GBK[13559] := 16#94D9;
   // UNICODE_TO_GBK[13560] := 16#65AF;
   // UNICODE_TO_GBK[13561] := 16#CBB9;
   // UNICODE_TO_GBK[13562] := 16#65B0;
   // UNICODE_TO_GBK[13563] := 16#D0C2;
   // UNICODE_TO_GBK[13564] := 16#65B1;
   // UNICODE_TO_GBK[13565] := 16#94DA;
   // UNICODE_TO_GBK[13566] := 16#65B2;
   // UNICODE_TO_GBK[13567] := 16#94DB;
   // UNICODE_TO_GBK[13568] := 16#65B3;
   // UNICODE_TO_GBK[13569] := 16#94DC;
   // UNICODE_TO_GBK[13570] := 16#65B4;
   // UNICODE_TO_GBK[13571] := 16#94DD;
   // UNICODE_TO_GBK[13572] := 16#65B5;
   // UNICODE_TO_GBK[13573] := 16#94DE;
   // UNICODE_TO_GBK[13574] := 16#65B6;
   // UNICODE_TO_GBK[13575] := 16#94DF;
   // UNICODE_TO_GBK[13576] := 16#65B7;
   // UNICODE_TO_GBK[13577] := 16#94E0;
   // UNICODE_TO_GBK[13578] := 16#65B8;
   // UNICODE_TO_GBK[13579] := 16#94E1;
   // UNICODE_TO_GBK[13580] := 16#65B9;
   // UNICODE_TO_GBK[13581] := 16#B7BD;
   // UNICODE_TO_GBK[13582] := 16#65BA;
   // UNICODE_TO_GBK[13583] := 16#94E2;
   // UNICODE_TO_GBK[13584] := 16#65BB;
   // UNICODE_TO_GBK[13585] := 16#94E3;
   // UNICODE_TO_GBK[13586] := 16#65BC;
   // UNICODE_TO_GBK[13587] := 16#ECB6;
   // UNICODE_TO_GBK[13588] := 16#65BD;
   // UNICODE_TO_GBK[13589] := 16#CAA9;
   // UNICODE_TO_GBK[13590] := 16#65BE;
   // UNICODE_TO_GBK[13591] := 16#94E4;
   // UNICODE_TO_GBK[13592] := 16#65BF;
   // UNICODE_TO_GBK[13593] := 16#94E5;
   // UNICODE_TO_GBK[13594] := 16#65C0;
   // UNICODE_TO_GBK[13595] := 16#94E6;
   // UNICODE_TO_GBK[13596] := 16#65C1;
   // UNICODE_TO_GBK[13597] := 16#C5D4;
   // UNICODE_TO_GBK[13598] := 16#65C2;
   // UNICODE_TO_GBK[13599] := 16#94E7;
   // UNICODE_TO_GBK[13600] := 16#65C3;
   // UNICODE_TO_GBK[13601] := 16#ECB9;
   // UNICODE_TO_GBK[13602] := 16#65C4;
   // UNICODE_TO_GBK[13603] := 16#ECB8;
   // UNICODE_TO_GBK[13604] := 16#65C5;
   // UNICODE_TO_GBK[13605] := 16#C2C3;
   // UNICODE_TO_GBK[13606] := 16#65C6;
   // UNICODE_TO_GBK[13607] := 16#ECB7;
   // UNICODE_TO_GBK[13608] := 16#65C7;
   // UNICODE_TO_GBK[13609] := 16#94E8;
   // UNICODE_TO_GBK[13610] := 16#65C8;
   // UNICODE_TO_GBK[13611] := 16#94E9;
   // UNICODE_TO_GBK[13612] := 16#65C9;
   // UNICODE_TO_GBK[13613] := 16#94EA;
   // UNICODE_TO_GBK[13614] := 16#65CA;
   // UNICODE_TO_GBK[13615] := 16#94EB;
   // UNICODE_TO_GBK[13616] := 16#65CB;
   // UNICODE_TO_GBK[13617] := 16#D0FD;
   // UNICODE_TO_GBK[13618] := 16#65CC;
   // UNICODE_TO_GBK[13619] := 16#ECBA;
   // UNICODE_TO_GBK[13620] := 16#65CD;
   // UNICODE_TO_GBK[13621] := 16#94EC;
   // UNICODE_TO_GBK[13622] := 16#65CE;
   // UNICODE_TO_GBK[13623] := 16#ECBB;
   // UNICODE_TO_GBK[13624] := 16#65CF;
   // UNICODE_TO_GBK[13625] := 16#D7E5;
   // UNICODE_TO_GBK[13626] := 16#65D0;
   // UNICODE_TO_GBK[13627] := 16#94ED;
   // UNICODE_TO_GBK[13628] := 16#65D1;
   // UNICODE_TO_GBK[13629] := 16#94EE;
   // UNICODE_TO_GBK[13630] := 16#65D2;
   // UNICODE_TO_GBK[13631] := 16#ECBC;
   // UNICODE_TO_GBK[13632] := 16#65D3;
   // UNICODE_TO_GBK[13633] := 16#94EF;
   // UNICODE_TO_GBK[13634] := 16#65D4;
   // UNICODE_TO_GBK[13635] := 16#94F0;
   // UNICODE_TO_GBK[13636] := 16#65D5;
   // UNICODE_TO_GBK[13637] := 16#94F1;
   // UNICODE_TO_GBK[13638] := 16#65D6;
   // UNICODE_TO_GBK[13639] := 16#ECBD;
   // UNICODE_TO_GBK[13640] := 16#65D7;
   // UNICODE_TO_GBK[13641] := 16#C6EC;
   // UNICODE_TO_GBK[13642] := 16#65D8;
   // UNICODE_TO_GBK[13643] := 16#94F2;
   // UNICODE_TO_GBK[13644] := 16#65D9;
   // UNICODE_TO_GBK[13645] := 16#94F3;
   // UNICODE_TO_GBK[13646] := 16#65DA;
   // UNICODE_TO_GBK[13647] := 16#94F4;
   // UNICODE_TO_GBK[13648] := 16#65DB;
   // UNICODE_TO_GBK[13649] := 16#94F5;
   // UNICODE_TO_GBK[13650] := 16#65DC;
   // UNICODE_TO_GBK[13651] := 16#94F6;
   // UNICODE_TO_GBK[13652] := 16#65DD;
   // UNICODE_TO_GBK[13653] := 16#94F7;
   // UNICODE_TO_GBK[13654] := 16#65DE;
   // UNICODE_TO_GBK[13655] := 16#94F8;
   // UNICODE_TO_GBK[13656] := 16#65DF;
   // UNICODE_TO_GBK[13657] := 16#94F9;
   // UNICODE_TO_GBK[13658] := 16#65E0;
   // UNICODE_TO_GBK[13659] := 16#CEDE;
   // UNICODE_TO_GBK[13660] := 16#65E1;
   // UNICODE_TO_GBK[13661] := 16#94FA;
   // UNICODE_TO_GBK[13662] := 16#65E2;
   // UNICODE_TO_GBK[13663] := 16#BCC8;
   // UNICODE_TO_GBK[13664] := 16#65E3;
   // UNICODE_TO_GBK[13665] := 16#94FB;
   // UNICODE_TO_GBK[13666] := 16#65E4;
   // UNICODE_TO_GBK[13667] := 16#94FC;
   // UNICODE_TO_GBK[13668] := 16#65E5;
   // UNICODE_TO_GBK[13669] := 16#C8D5;
   // UNICODE_TO_GBK[13670] := 16#65E6;
   // UNICODE_TO_GBK[13671] := 16#B5A9;
   // UNICODE_TO_GBK[13672] := 16#65E7;
   // UNICODE_TO_GBK[13673] := 16#BEC9;
   // UNICODE_TO_GBK[13674] := 16#65E8;
   // UNICODE_TO_GBK[13675] := 16#D6BC;
   // UNICODE_TO_GBK[13676] := 16#65E9;
   // UNICODE_TO_GBK[13677] := 16#D4E7;
   // UNICODE_TO_GBK[13678] := 16#65EA;
   // UNICODE_TO_GBK[13679] := 16#94FD;
   // UNICODE_TO_GBK[13680] := 16#65EB;
   // UNICODE_TO_GBK[13681] := 16#94FE;
   // UNICODE_TO_GBK[13682] := 16#65EC;
   // UNICODE_TO_GBK[13683] := 16#D1AE;
   // UNICODE_TO_GBK[13684] := 16#65ED;
   // UNICODE_TO_GBK[13685] := 16#D0F1;
   // UNICODE_TO_GBK[13686] := 16#65EE;
   // UNICODE_TO_GBK[13687] := 16#EAB8;
   // UNICODE_TO_GBK[13688] := 16#65EF;
   // UNICODE_TO_GBK[13689] := 16#EAB9;
   // UNICODE_TO_GBK[13690] := 16#65F0;
   // UNICODE_TO_GBK[13691] := 16#EABA;
   // UNICODE_TO_GBK[13692] := 16#65F1;
   // UNICODE_TO_GBK[13693] := 16#BAB5;
   // UNICODE_TO_GBK[13694] := 16#65F2;
   // UNICODE_TO_GBK[13695] := 16#9540;
   // UNICODE_TO_GBK[13696] := 16#65F3;
   // UNICODE_TO_GBK[13697] := 16#9541;
   // UNICODE_TO_GBK[13698] := 16#65F4;
   // UNICODE_TO_GBK[13699] := 16#9542;
   // UNICODE_TO_GBK[13700] := 16#65F5;
   // UNICODE_TO_GBK[13701] := 16#9543;
   // UNICODE_TO_GBK[13702] := 16#65F6;
   // UNICODE_TO_GBK[13703] := 16#CAB1;
   // UNICODE_TO_GBK[13704] := 16#65F7;
   // UNICODE_TO_GBK[13705] := 16#BFF5;
   // UNICODE_TO_GBK[13706] := 16#65F8;
   // UNICODE_TO_GBK[13707] := 16#9544;
   // UNICODE_TO_GBK[13708] := 16#65F9;
   // UNICODE_TO_GBK[13709] := 16#9545;
   // UNICODE_TO_GBK[13710] := 16#65FA;
   // UNICODE_TO_GBK[13711] := 16#CDFA;
   // UNICODE_TO_GBK[13712] := 16#65FB;
   // UNICODE_TO_GBK[13713] := 16#9546;
   // UNICODE_TO_GBK[13714] := 16#65FC;
   // UNICODE_TO_GBK[13715] := 16#9547;
   // UNICODE_TO_GBK[13716] := 16#65FD;
   // UNICODE_TO_GBK[13717] := 16#9548;
   // UNICODE_TO_GBK[13718] := 16#65FE;
   // UNICODE_TO_GBK[13719] := 16#9549;
   // UNICODE_TO_GBK[13720] := 16#65FF;
   // UNICODE_TO_GBK[13721] := 16#954A;
   // UNICODE_TO_GBK[13722] := 16#6600;
   // UNICODE_TO_GBK[13723] := 16#EAC0;
   // UNICODE_TO_GBK[13724] := 16#6601;
   // UNICODE_TO_GBK[13725] := 16#954B;
   // UNICODE_TO_GBK[13726] := 16#6602;
   // UNICODE_TO_GBK[13727] := 16#B0BA;
   // UNICODE_TO_GBK[13728] := 16#6603;
   // UNICODE_TO_GBK[13729] := 16#EABE;
   // UNICODE_TO_GBK[13730] := 16#6604;
   // UNICODE_TO_GBK[13731] := 16#954C;
   // UNICODE_TO_GBK[13732] := 16#6605;
   // UNICODE_TO_GBK[13733] := 16#954D;
   // UNICODE_TO_GBK[13734] := 16#6606;
   // UNICODE_TO_GBK[13735] := 16#C0A5;
   // UNICODE_TO_GBK[13736] := 16#6607;
   // UNICODE_TO_GBK[13737] := 16#954E;
   // UNICODE_TO_GBK[13738] := 16#6608;
   // UNICODE_TO_GBK[13739] := 16#954F;
   // UNICODE_TO_GBK[13740] := 16#6609;
   // UNICODE_TO_GBK[13741] := 16#9550;
   // UNICODE_TO_GBK[13742] := 16#660A;
   // UNICODE_TO_GBK[13743] := 16#EABB;
   // UNICODE_TO_GBK[13744] := 16#660B;
   // UNICODE_TO_GBK[13745] := 16#9551;
   // UNICODE_TO_GBK[13746] := 16#660C;
   // UNICODE_TO_GBK[13747] := 16#B2FD;
   // UNICODE_TO_GBK[13748] := 16#660D;
   // UNICODE_TO_GBK[13749] := 16#9552;
   // UNICODE_TO_GBK[13750] := 16#660E;
   // UNICODE_TO_GBK[13751] := 16#C3F7;
   // UNICODE_TO_GBK[13752] := 16#660F;
   // UNICODE_TO_GBK[13753] := 16#BBE8;
   // UNICODE_TO_GBK[13754] := 16#6610;
   // UNICODE_TO_GBK[13755] := 16#9553;
   // UNICODE_TO_GBK[13756] := 16#6611;
   // UNICODE_TO_GBK[13757] := 16#9554;
   // UNICODE_TO_GBK[13758] := 16#6612;
   // UNICODE_TO_GBK[13759] := 16#9555;
   // UNICODE_TO_GBK[13760] := 16#6613;
   // UNICODE_TO_GBK[13761] := 16#D2D7;
   // UNICODE_TO_GBK[13762] := 16#6614;
   // UNICODE_TO_GBK[13763] := 16#CEF4;
   // UNICODE_TO_GBK[13764] := 16#6615;
   // UNICODE_TO_GBK[13765] := 16#EABF;
   // UNICODE_TO_GBK[13766] := 16#6616;
   // UNICODE_TO_GBK[13767] := 16#9556;
   // UNICODE_TO_GBK[13768] := 16#6617;
   // UNICODE_TO_GBK[13769] := 16#9557;
   // UNICODE_TO_GBK[13770] := 16#6618;
   // UNICODE_TO_GBK[13771] := 16#9558;
   // UNICODE_TO_GBK[13772] := 16#6619;
   // UNICODE_TO_GBK[13773] := 16#EABC;
   // UNICODE_TO_GBK[13774] := 16#661A;
   // UNICODE_TO_GBK[13775] := 16#9559;
   // UNICODE_TO_GBK[13776] := 16#661B;
   // UNICODE_TO_GBK[13777] := 16#955A;
   // UNICODE_TO_GBK[13778] := 16#661C;
   // UNICODE_TO_GBK[13779] := 16#955B;
   // UNICODE_TO_GBK[13780] := 16#661D;
   // UNICODE_TO_GBK[13781] := 16#EAC3;
   // UNICODE_TO_GBK[13782] := 16#661E;
   // UNICODE_TO_GBK[13783] := 16#955C;
   // UNICODE_TO_GBK[13784] := 16#661F;
   // UNICODE_TO_GBK[13785] := 16#D0C7;
   // UNICODE_TO_GBK[13786] := 16#6620;
   // UNICODE_TO_GBK[13787] := 16#D3B3;
   // UNICODE_TO_GBK[13788] := 16#6621;
   // UNICODE_TO_GBK[13789] := 16#955D;
   // UNICODE_TO_GBK[13790] := 16#6622;
   // UNICODE_TO_GBK[13791] := 16#955E;
   // UNICODE_TO_GBK[13792] := 16#6623;
   // UNICODE_TO_GBK[13793] := 16#955F;
   // UNICODE_TO_GBK[13794] := 16#6624;
   // UNICODE_TO_GBK[13795] := 16#9560;
   // UNICODE_TO_GBK[13796] := 16#6625;
   // UNICODE_TO_GBK[13797] := 16#B4BA;
   // UNICODE_TO_GBK[13798] := 16#6626;
   // UNICODE_TO_GBK[13799] := 16#9561;
   // UNICODE_TO_GBK[13800] := 16#6627;
   // UNICODE_TO_GBK[13801] := 16#C3C1;
   // UNICODE_TO_GBK[13802] := 16#6628;
   // UNICODE_TO_GBK[13803] := 16#D7F2;
   // UNICODE_TO_GBK[13804] := 16#6629;
   // UNICODE_TO_GBK[13805] := 16#9562;
   // UNICODE_TO_GBK[13806] := 16#662A;
   // UNICODE_TO_GBK[13807] := 16#9563;
   // UNICODE_TO_GBK[13808] := 16#662B;
   // UNICODE_TO_GBK[13809] := 16#9564;
   // UNICODE_TO_GBK[13810] := 16#662C;
   // UNICODE_TO_GBK[13811] := 16#9565;
   // UNICODE_TO_GBK[13812] := 16#662D;
   // UNICODE_TO_GBK[13813] := 16#D5D1;
   // UNICODE_TO_GBK[13814] := 16#662E;
   // UNICODE_TO_GBK[13815] := 16#9566;
   // UNICODE_TO_GBK[13816] := 16#662F;
   // UNICODE_TO_GBK[13817] := 16#CAC7;
   // UNICODE_TO_GBK[13818] := 16#6630;
   // UNICODE_TO_GBK[13819] := 16#9567;
   // UNICODE_TO_GBK[13820] := 16#6631;
   // UNICODE_TO_GBK[13821] := 16#EAC5;
   // UNICODE_TO_GBK[13822] := 16#6632;
   // UNICODE_TO_GBK[13823] := 16#9568;
   // UNICODE_TO_GBK[13824] := 16#6633;
   // UNICODE_TO_GBK[13825] := 16#9569;
   // UNICODE_TO_GBK[13826] := 16#6634;
   // UNICODE_TO_GBK[13827] := 16#EAC4;
   // UNICODE_TO_GBK[13828] := 16#6635;
   // UNICODE_TO_GBK[13829] := 16#EAC7;
   // UNICODE_TO_GBK[13830] := 16#6636;
   // UNICODE_TO_GBK[13831] := 16#EAC6;
   // UNICODE_TO_GBK[13832] := 16#6637;
   // UNICODE_TO_GBK[13833] := 16#956A;
   // UNICODE_TO_GBK[13834] := 16#6638;
   // UNICODE_TO_GBK[13835] := 16#956B;
   // UNICODE_TO_GBK[13836] := 16#6639;
   // UNICODE_TO_GBK[13837] := 16#956C;
   // UNICODE_TO_GBK[13838] := 16#663A;
   // UNICODE_TO_GBK[13839] := 16#956D;
   // UNICODE_TO_GBK[13840] := 16#663B;
   // UNICODE_TO_GBK[13841] := 16#956E;
   // UNICODE_TO_GBK[13842] := 16#663C;
   // UNICODE_TO_GBK[13843] := 16#D6E7;
   // UNICODE_TO_GBK[13844] := 16#663D;
   // UNICODE_TO_GBK[13845] := 16#956F;
   // UNICODE_TO_GBK[13846] := 16#663E;
   // UNICODE_TO_GBK[13847] := 16#CFD4;
   // UNICODE_TO_GBK[13848] := 16#663F;
   // UNICODE_TO_GBK[13849] := 16#9570;
   // UNICODE_TO_GBK[13850] := 16#6640;
   // UNICODE_TO_GBK[13851] := 16#9571;
   // UNICODE_TO_GBK[13852] := 16#6641;
   // UNICODE_TO_GBK[13853] := 16#EACB;
   // UNICODE_TO_GBK[13854] := 16#6642;
   // UNICODE_TO_GBK[13855] := 16#9572;
   // UNICODE_TO_GBK[13856] := 16#6643;
   // UNICODE_TO_GBK[13857] := 16#BBCE;
   // UNICODE_TO_GBK[13858] := 16#6644;
   // UNICODE_TO_GBK[13859] := 16#9573;
   // UNICODE_TO_GBK[13860] := 16#6645;
   // UNICODE_TO_GBK[13861] := 16#9574;
   // UNICODE_TO_GBK[13862] := 16#6646;
   // UNICODE_TO_GBK[13863] := 16#9575;
   // UNICODE_TO_GBK[13864] := 16#6647;
   // UNICODE_TO_GBK[13865] := 16#9576;
   // UNICODE_TO_GBK[13866] := 16#6648;
   // UNICODE_TO_GBK[13867] := 16#9577;
   // UNICODE_TO_GBK[13868] := 16#6649;
   // UNICODE_TO_GBK[13869] := 16#9578;
   // UNICODE_TO_GBK[13870] := 16#664A;
   // UNICODE_TO_GBK[13871] := 16#9579;
   // UNICODE_TO_GBK[13872] := 16#664B;
   // UNICODE_TO_GBK[13873] := 16#BDFA;
   // UNICODE_TO_GBK[13874] := 16#664C;
   // UNICODE_TO_GBK[13875] := 16#C9CE;
   // UNICODE_TO_GBK[13876] := 16#664D;
   // UNICODE_TO_GBK[13877] := 16#957A;
   // UNICODE_TO_GBK[13878] := 16#664E;
   // UNICODE_TO_GBK[13879] := 16#957B;
   // UNICODE_TO_GBK[13880] := 16#664F;
   // UNICODE_TO_GBK[13881] := 16#EACC;
   // UNICODE_TO_GBK[13882] := 16#6650;
   // UNICODE_TO_GBK[13883] := 16#957C;
   // UNICODE_TO_GBK[13884] := 16#6651;
   // UNICODE_TO_GBK[13885] := 16#957D;
   // UNICODE_TO_GBK[13886] := 16#6652;
   // UNICODE_TO_GBK[13887] := 16#C9B9;
   // UNICODE_TO_GBK[13888] := 16#6653;
   // UNICODE_TO_GBK[13889] := 16#CFFE;
   // UNICODE_TO_GBK[13890] := 16#6654;
   // UNICODE_TO_GBK[13891] := 16#EACA;
   // UNICODE_TO_GBK[13892] := 16#6655;
   // UNICODE_TO_GBK[13893] := 16#D4CE;
   // UNICODE_TO_GBK[13894] := 16#6656;
   // UNICODE_TO_GBK[13895] := 16#EACD;
   // UNICODE_TO_GBK[13896] := 16#6657;
   // UNICODE_TO_GBK[13897] := 16#EACF;
   // UNICODE_TO_GBK[13898] := 16#6658;
   // UNICODE_TO_GBK[13899] := 16#957E;
   // UNICODE_TO_GBK[13900] := 16#6659;
   // UNICODE_TO_GBK[13901] := 16#9580;
   // UNICODE_TO_GBK[13902] := 16#665A;
   // UNICODE_TO_GBK[13903] := 16#CDED;
   // UNICODE_TO_GBK[13904] := 16#665B;
   // UNICODE_TO_GBK[13905] := 16#9581;
   // UNICODE_TO_GBK[13906] := 16#665C;
   // UNICODE_TO_GBK[13907] := 16#9582;
   // UNICODE_TO_GBK[13908] := 16#665D;
   // UNICODE_TO_GBK[13909] := 16#9583;
   // UNICODE_TO_GBK[13910] := 16#665E;
   // UNICODE_TO_GBK[13911] := 16#9584;
   // UNICODE_TO_GBK[13912] := 16#665F;
   // UNICODE_TO_GBK[13913] := 16#EAC9;
   // UNICODE_TO_GBK[13914] := 16#6660;
   // UNICODE_TO_GBK[13915] := 16#9585;
   // UNICODE_TO_GBK[13916] := 16#6661;
   // UNICODE_TO_GBK[13917] := 16#EACE;
   // UNICODE_TO_GBK[13918] := 16#6662;
   // UNICODE_TO_GBK[13919] := 16#9586;
   // UNICODE_TO_GBK[13920] := 16#6663;
   // UNICODE_TO_GBK[13921] := 16#9587;
   // UNICODE_TO_GBK[13922] := 16#6664;
   // UNICODE_TO_GBK[13923] := 16#CEEE;
   // UNICODE_TO_GBK[13924] := 16#6665;
   // UNICODE_TO_GBK[13925] := 16#9588;
   // UNICODE_TO_GBK[13926] := 16#6666;
   // UNICODE_TO_GBK[13927] := 16#BBDE;
   // UNICODE_TO_GBK[13928] := 16#6667;
   // UNICODE_TO_GBK[13929] := 16#9589;
   // UNICODE_TO_GBK[13930] := 16#6668;
   // UNICODE_TO_GBK[13931] := 16#B3BF;
   // UNICODE_TO_GBK[13932] := 16#6669;
   // UNICODE_TO_GBK[13933] := 16#958A;
   // UNICODE_TO_GBK[13934] := 16#666A;
   // UNICODE_TO_GBK[13935] := 16#958B;
   // UNICODE_TO_GBK[13936] := 16#666B;
   // UNICODE_TO_GBK[13937] := 16#958C;
   // UNICODE_TO_GBK[13938] := 16#666C;
   // UNICODE_TO_GBK[13939] := 16#958D;
   // UNICODE_TO_GBK[13940] := 16#666D;
   // UNICODE_TO_GBK[13941] := 16#958E;
   // UNICODE_TO_GBK[13942] := 16#666E;
   // UNICODE_TO_GBK[13943] := 16#C6D5;
   // UNICODE_TO_GBK[13944] := 16#666F;
   // UNICODE_TO_GBK[13945] := 16#BEB0;
   // UNICODE_TO_GBK[13946] := 16#6670;
   // UNICODE_TO_GBK[13947] := 16#CEFA;
   // UNICODE_TO_GBK[13948] := 16#6671;
   // UNICODE_TO_GBK[13949] := 16#958F;
   // UNICODE_TO_GBK[13950] := 16#6672;
   // UNICODE_TO_GBK[13951] := 16#9590;
   // UNICODE_TO_GBK[13952] := 16#6673;
   // UNICODE_TO_GBK[13953] := 16#9591;
   // UNICODE_TO_GBK[13954] := 16#6674;
   // UNICODE_TO_GBK[13955] := 16#C7E7;
   // UNICODE_TO_GBK[13956] := 16#6675;
   // UNICODE_TO_GBK[13957] := 16#9592;
   // UNICODE_TO_GBK[13958] := 16#6676;
   // UNICODE_TO_GBK[13959] := 16#BEA7;
   // UNICODE_TO_GBK[13960] := 16#6677;
   // UNICODE_TO_GBK[13961] := 16#EAD0;
   // UNICODE_TO_GBK[13962] := 16#6678;
   // UNICODE_TO_GBK[13963] := 16#9593;
   // UNICODE_TO_GBK[13964] := 16#6679;
   // UNICODE_TO_GBK[13965] := 16#9594;
   // UNICODE_TO_GBK[13966] := 16#667A;
   // UNICODE_TO_GBK[13967] := 16#D6C7;
   // UNICODE_TO_GBK[13968] := 16#667B;
   // UNICODE_TO_GBK[13969] := 16#9595;
   // UNICODE_TO_GBK[13970] := 16#667C;
   // UNICODE_TO_GBK[13971] := 16#9596;
   // UNICODE_TO_GBK[13972] := 16#667D;
   // UNICODE_TO_GBK[13973] := 16#9597;
   // UNICODE_TO_GBK[13974] := 16#667E;
   // UNICODE_TO_GBK[13975] := 16#C1C0;
   // UNICODE_TO_GBK[13976] := 16#667F;
   // UNICODE_TO_GBK[13977] := 16#9598;
   // UNICODE_TO_GBK[13978] := 16#6680;
   // UNICODE_TO_GBK[13979] := 16#9599;
   // UNICODE_TO_GBK[13980] := 16#6681;
   // UNICODE_TO_GBK[13981] := 16#959A;
   // UNICODE_TO_GBK[13982] := 16#6682;
   // UNICODE_TO_GBK[13983] := 16#D4DD;
   // UNICODE_TO_GBK[13984] := 16#6683;
   // UNICODE_TO_GBK[13985] := 16#959B;
   // UNICODE_TO_GBK[13986] := 16#6684;
   // UNICODE_TO_GBK[13987] := 16#EAD1;
   // UNICODE_TO_GBK[13988] := 16#6685;
   // UNICODE_TO_GBK[13989] := 16#959C;
   // UNICODE_TO_GBK[13990] := 16#6686;
   // UNICODE_TO_GBK[13991] := 16#959D;
   // UNICODE_TO_GBK[13992] := 16#6687;
   // UNICODE_TO_GBK[13993] := 16#CFBE;
   // UNICODE_TO_GBK[13994] := 16#6688;
   // UNICODE_TO_GBK[13995] := 16#959E;
   // UNICODE_TO_GBK[13996] := 16#6689;
   // UNICODE_TO_GBK[13997] := 16#959F;
   // UNICODE_TO_GBK[13998] := 16#668A;
   // UNICODE_TO_GBK[13999] := 16#95A0;
   // UNICODE_TO_GBK[14000] := 16#668B;
   // UNICODE_TO_GBK[14001] := 16#95A1;
   // UNICODE_TO_GBK[14002] := 16#668C;
   // UNICODE_TO_GBK[14003] := 16#EAD2;
   // UNICODE_TO_GBK[14004] := 16#668D;
   // UNICODE_TO_GBK[14005] := 16#95A2;
   // UNICODE_TO_GBK[14006] := 16#668E;
   // UNICODE_TO_GBK[14007] := 16#95A3;
   // UNICODE_TO_GBK[14008] := 16#668F;
   // UNICODE_TO_GBK[14009] := 16#95A4;
   // UNICODE_TO_GBK[14010] := 16#6690;
   // UNICODE_TO_GBK[14011] := 16#95A5;
   // UNICODE_TO_GBK[14012] := 16#6691;
   // UNICODE_TO_GBK[14013] := 16#CAEE;
   // UNICODE_TO_GBK[14014] := 16#6692;
   // UNICODE_TO_GBK[14015] := 16#95A6;
   // UNICODE_TO_GBK[14016] := 16#6693;
   // UNICODE_TO_GBK[14017] := 16#95A7;
   // UNICODE_TO_GBK[14018] := 16#6694;
   // UNICODE_TO_GBK[14019] := 16#95A8;
   // UNICODE_TO_GBK[14020] := 16#6695;
   // UNICODE_TO_GBK[14021] := 16#95A9;
   // UNICODE_TO_GBK[14022] := 16#6696;
   // UNICODE_TO_GBK[14023] := 16#C5AF;
   // UNICODE_TO_GBK[14024] := 16#6697;
   // UNICODE_TO_GBK[14025] := 16#B0B5;
   // UNICODE_TO_GBK[14026] := 16#6698;
   // UNICODE_TO_GBK[14027] := 16#95AA;
   // UNICODE_TO_GBK[14028] := 16#6699;
   // UNICODE_TO_GBK[14029] := 16#95AB;
   // UNICODE_TO_GBK[14030] := 16#669A;
   // UNICODE_TO_GBK[14031] := 16#95AC;
   // UNICODE_TO_GBK[14032] := 16#669B;
   // UNICODE_TO_GBK[14033] := 16#95AD;
   // UNICODE_TO_GBK[14034] := 16#669C;
   // UNICODE_TO_GBK[14035] := 16#95AE;
   // UNICODE_TO_GBK[14036] := 16#669D;
   // UNICODE_TO_GBK[14037] := 16#EAD4;
   // UNICODE_TO_GBK[14038] := 16#669E;
   // UNICODE_TO_GBK[14039] := 16#95AF;
   // UNICODE_TO_GBK[14040] := 16#669F;
   // UNICODE_TO_GBK[14041] := 16#95B0;
   // UNICODE_TO_GBK[14042] := 16#66A0;
   // UNICODE_TO_GBK[14043] := 16#95B1;
   // UNICODE_TO_GBK[14044] := 16#66A1;
   // UNICODE_TO_GBK[14045] := 16#95B2;
   // UNICODE_TO_GBK[14046] := 16#66A2;
   // UNICODE_TO_GBK[14047] := 16#95B3;
   // UNICODE_TO_GBK[14048] := 16#66A3;
   // UNICODE_TO_GBK[14049] := 16#95B4;
   // UNICODE_TO_GBK[14050] := 16#66A4;
   // UNICODE_TO_GBK[14051] := 16#95B5;
   // UNICODE_TO_GBK[14052] := 16#66A5;
   // UNICODE_TO_GBK[14053] := 16#95B6;
   // UNICODE_TO_GBK[14054] := 16#66A6;
   // UNICODE_TO_GBK[14055] := 16#95B7;
   // UNICODE_TO_GBK[14056] := 16#66A7;
   // UNICODE_TO_GBK[14057] := 16#EAD3;
   // UNICODE_TO_GBK[14058] := 16#66A8;
   // UNICODE_TO_GBK[14059] := 16#F4DF;
   // UNICODE_TO_GBK[14060] := 16#66A9;
   // UNICODE_TO_GBK[14061] := 16#95B8;
   // UNICODE_TO_GBK[14062] := 16#66AA;
   // UNICODE_TO_GBK[14063] := 16#95B9;
   // UNICODE_TO_GBK[14064] := 16#66AB;
   // UNICODE_TO_GBK[14065] := 16#95BA;
   // UNICODE_TO_GBK[14066] := 16#66AC;
   // UNICODE_TO_GBK[14067] := 16#95BB;
   // UNICODE_TO_GBK[14068] := 16#66AD;
   // UNICODE_TO_GBK[14069] := 16#95BC;
   // UNICODE_TO_GBK[14070] := 16#66AE;
   // UNICODE_TO_GBK[14071] := 16#C4BA;
   // UNICODE_TO_GBK[14072] := 16#66AF;
   // UNICODE_TO_GBK[14073] := 16#95BD;
   // UNICODE_TO_GBK[14074] := 16#66B0;
   // UNICODE_TO_GBK[14075] := 16#95BE;
   // UNICODE_TO_GBK[14076] := 16#66B1;
   // UNICODE_TO_GBK[14077] := 16#95BF;
   // UNICODE_TO_GBK[14078] := 16#66B2;
   // UNICODE_TO_GBK[14079] := 16#95C0;
   // UNICODE_TO_GBK[14080] := 16#66B3;
   // UNICODE_TO_GBK[14081] := 16#95C1;
   // UNICODE_TO_GBK[14082] := 16#66B4;
   // UNICODE_TO_GBK[14083] := 16#B1A9;
   // UNICODE_TO_GBK[14084] := 16#66B5;
   // UNICODE_TO_GBK[14085] := 16#95C2;
   // UNICODE_TO_GBK[14086] := 16#66B6;
   // UNICODE_TO_GBK[14087] := 16#95C3;
   // UNICODE_TO_GBK[14088] := 16#66B7;
   // UNICODE_TO_GBK[14089] := 16#95C4;
   // UNICODE_TO_GBK[14090] := 16#66B8;
   // UNICODE_TO_GBK[14091] := 16#95C5;
   // UNICODE_TO_GBK[14092] := 16#66B9;
   // UNICODE_TO_GBK[14093] := 16#E5DF;
   // UNICODE_TO_GBK[14094] := 16#66BA;
   // UNICODE_TO_GBK[14095] := 16#95C6;
   // UNICODE_TO_GBK[14096] := 16#66BB;
   // UNICODE_TO_GBK[14097] := 16#95C7;
   // UNICODE_TO_GBK[14098] := 16#66BC;
   // UNICODE_TO_GBK[14099] := 16#95C8;
   // UNICODE_TO_GBK[14100] := 16#66BD;
   // UNICODE_TO_GBK[14101] := 16#95C9;
   // UNICODE_TO_GBK[14102] := 16#66BE;
   // UNICODE_TO_GBK[14103] := 16#EAD5;
   // UNICODE_TO_GBK[14104] := 16#66BF;
   // UNICODE_TO_GBK[14105] := 16#95CA;
   // UNICODE_TO_GBK[14106] := 16#66C0;
   // UNICODE_TO_GBK[14107] := 16#95CB;
   // UNICODE_TO_GBK[14108] := 16#66C1;
   // UNICODE_TO_GBK[14109] := 16#95CC;
   // UNICODE_TO_GBK[14110] := 16#66C2;
   // UNICODE_TO_GBK[14111] := 16#95CD;
   // UNICODE_TO_GBK[14112] := 16#66C3;
   // UNICODE_TO_GBK[14113] := 16#95CE;
   // UNICODE_TO_GBK[14114] := 16#66C4;
   // UNICODE_TO_GBK[14115] := 16#95CF;
   // UNICODE_TO_GBK[14116] := 16#66C5;
   // UNICODE_TO_GBK[14117] := 16#95D0;
   // UNICODE_TO_GBK[14118] := 16#66C6;
   // UNICODE_TO_GBK[14119] := 16#95D1;
   // UNICODE_TO_GBK[14120] := 16#66C7;
   // UNICODE_TO_GBK[14121] := 16#95D2;
   // UNICODE_TO_GBK[14122] := 16#66C8;
   // UNICODE_TO_GBK[14123] := 16#95D3;
   // UNICODE_TO_GBK[14124] := 16#66C9;
   // UNICODE_TO_GBK[14125] := 16#95D4;
   // UNICODE_TO_GBK[14126] := 16#66CA;
   // UNICODE_TO_GBK[14127] := 16#95D5;
   // UNICODE_TO_GBK[14128] := 16#66CB;
   // UNICODE_TO_GBK[14129] := 16#95D6;
   // UNICODE_TO_GBK[14130] := 16#66CC;
   // UNICODE_TO_GBK[14131] := 16#95D7;
   // UNICODE_TO_GBK[14132] := 16#66CD;
   // UNICODE_TO_GBK[14133] := 16#95D8;
   // UNICODE_TO_GBK[14134] := 16#66CE;
   // UNICODE_TO_GBK[14135] := 16#95D9;
   // UNICODE_TO_GBK[14136] := 16#66CF;
   // UNICODE_TO_GBK[14137] := 16#95DA;
   // UNICODE_TO_GBK[14138] := 16#66D0;
   // UNICODE_TO_GBK[14139] := 16#95DB;
   // UNICODE_TO_GBK[14140] := 16#66D1;
   // UNICODE_TO_GBK[14141] := 16#95DC;
   // UNICODE_TO_GBK[14142] := 16#66D2;
   // UNICODE_TO_GBK[14143] := 16#95DD;
   // UNICODE_TO_GBK[14144] := 16#66D3;
   // UNICODE_TO_GBK[14145] := 16#95DE;
   // UNICODE_TO_GBK[14146] := 16#66D4;
   // UNICODE_TO_GBK[14147] := 16#95DF;
   // UNICODE_TO_GBK[14148] := 16#66D5;
   // UNICODE_TO_GBK[14149] := 16#95E0;
   // UNICODE_TO_GBK[14150] := 16#66D6;
   // UNICODE_TO_GBK[14151] := 16#95E1;
   // UNICODE_TO_GBK[14152] := 16#66D7;
   // UNICODE_TO_GBK[14153] := 16#95E2;
   // UNICODE_TO_GBK[14154] := 16#66D8;
   // UNICODE_TO_GBK[14155] := 16#95E3;
   // UNICODE_TO_GBK[14156] := 16#66D9;
   // UNICODE_TO_GBK[14157] := 16#CAEF;
   // UNICODE_TO_GBK[14158] := 16#66DA;
   // UNICODE_TO_GBK[14159] := 16#95E4;
   // UNICODE_TO_GBK[14160] := 16#66DB;
   // UNICODE_TO_GBK[14161] := 16#EAD6;
   // UNICODE_TO_GBK[14162] := 16#66DC;
   // UNICODE_TO_GBK[14163] := 16#EAD7;
   // UNICODE_TO_GBK[14164] := 16#66DD;
   // UNICODE_TO_GBK[14165] := 16#C6D8;
   // UNICODE_TO_GBK[14166] := 16#66DE;
   // UNICODE_TO_GBK[14167] := 16#95E5;
   // UNICODE_TO_GBK[14168] := 16#66DF;
   // UNICODE_TO_GBK[14169] := 16#95E6;
   // UNICODE_TO_GBK[14170] := 16#66E0;
   // UNICODE_TO_GBK[14171] := 16#95E7;
   // UNICODE_TO_GBK[14172] := 16#66E1;
   // UNICODE_TO_GBK[14173] := 16#95E8;
   // UNICODE_TO_GBK[14174] := 16#66E2;
   // UNICODE_TO_GBK[14175] := 16#95E9;
   // UNICODE_TO_GBK[14176] := 16#66E3;
   // UNICODE_TO_GBK[14177] := 16#95EA;
   // UNICODE_TO_GBK[14178] := 16#66E4;
   // UNICODE_TO_GBK[14179] := 16#95EB;
   // UNICODE_TO_GBK[14180] := 16#66E5;
   // UNICODE_TO_GBK[14181] := 16#95EC;
   // UNICODE_TO_GBK[14182] := 16#66E6;
   // UNICODE_TO_GBK[14183] := 16#EAD8;
   // UNICODE_TO_GBK[14184] := 16#66E7;
   // UNICODE_TO_GBK[14185] := 16#95ED;
   // UNICODE_TO_GBK[14186] := 16#66E8;
   // UNICODE_TO_GBK[14187] := 16#95EE;
   // UNICODE_TO_GBK[14188] := 16#66E9;
   // UNICODE_TO_GBK[14189] := 16#EAD9;
   // UNICODE_TO_GBK[14190] := 16#66EA;
   // UNICODE_TO_GBK[14191] := 16#95EF;
   // UNICODE_TO_GBK[14192] := 16#66EB;
   // UNICODE_TO_GBK[14193] := 16#95F0;
   // UNICODE_TO_GBK[14194] := 16#66EC;
   // UNICODE_TO_GBK[14195] := 16#95F1;
   // UNICODE_TO_GBK[14196] := 16#66ED;
   // UNICODE_TO_GBK[14197] := 16#95F2;
   // UNICODE_TO_GBK[14198] := 16#66EE;
   // UNICODE_TO_GBK[14199] := 16#95F3;
   // UNICODE_TO_GBK[14200] := 16#66EF;
   // UNICODE_TO_GBK[14201] := 16#95F4;
   // UNICODE_TO_GBK[14202] := 16#66F0;
   // UNICODE_TO_GBK[14203] := 16#D4BB;
   // UNICODE_TO_GBK[14204] := 16#66F1;
   // UNICODE_TO_GBK[14205] := 16#95F5;
   // UNICODE_TO_GBK[14206] := 16#66F2;
   // UNICODE_TO_GBK[14207] := 16#C7FA;
   // UNICODE_TO_GBK[14208] := 16#66F3;
   // UNICODE_TO_GBK[14209] := 16#D2B7;
   // UNICODE_TO_GBK[14210] := 16#66F4;
   // UNICODE_TO_GBK[14211] := 16#B8FC;
   // UNICODE_TO_GBK[14212] := 16#66F5;
   // UNICODE_TO_GBK[14213] := 16#95F6;
   // UNICODE_TO_GBK[14214] := 16#66F6;
   // UNICODE_TO_GBK[14215] := 16#95F7;
   // UNICODE_TO_GBK[14216] := 16#66F7;
   // UNICODE_TO_GBK[14217] := 16#EAC2;
   // UNICODE_TO_GBK[14218] := 16#66F8;
   // UNICODE_TO_GBK[14219] := 16#95F8;
   // UNICODE_TO_GBK[14220] := 16#66F9;
   // UNICODE_TO_GBK[14221] := 16#B2DC;
   // UNICODE_TO_GBK[14222] := 16#66FA;
   // UNICODE_TO_GBK[14223] := 16#95F9;
   // UNICODE_TO_GBK[14224] := 16#66FB;
   // UNICODE_TO_GBK[14225] := 16#95FA;
   // UNICODE_TO_GBK[14226] := 16#66FC;
   // UNICODE_TO_GBK[14227] := 16#C2FC;
   // UNICODE_TO_GBK[14228] := 16#66FD;
   // UNICODE_TO_GBK[14229] := 16#95FB;
   // UNICODE_TO_GBK[14230] := 16#66FE;
   // UNICODE_TO_GBK[14231] := 16#D4F8;
   // UNICODE_TO_GBK[14232] := 16#66FF;
   // UNICODE_TO_GBK[14233] := 16#CCE6;
   // UNICODE_TO_GBK[14234] := 16#6700;
   // UNICODE_TO_GBK[14235] := 16#D7EE;
   // UNICODE_TO_GBK[14236] := 16#6701;
   // UNICODE_TO_GBK[14237] := 16#95FC;
   // UNICODE_TO_GBK[14238] := 16#6702;
   // UNICODE_TO_GBK[14239] := 16#95FD;
   // UNICODE_TO_GBK[14240] := 16#6703;
   // UNICODE_TO_GBK[14241] := 16#95FE;
   // UNICODE_TO_GBK[14242] := 16#6704;
   // UNICODE_TO_GBK[14243] := 16#9640;
   // UNICODE_TO_GBK[14244] := 16#6705;
   // UNICODE_TO_GBK[14245] := 16#9641;
   // UNICODE_TO_GBK[14246] := 16#6706;
   // UNICODE_TO_GBK[14247] := 16#9642;
   // UNICODE_TO_GBK[14248] := 16#6707;
   // UNICODE_TO_GBK[14249] := 16#9643;
   // UNICODE_TO_GBK[14250] := 16#6708;
   // UNICODE_TO_GBK[14251] := 16#D4C2;
   // UNICODE_TO_GBK[14252] := 16#6709;
   // UNICODE_TO_GBK[14253] := 16#D3D0;
   // UNICODE_TO_GBK[14254] := 16#670A;
   // UNICODE_TO_GBK[14255] := 16#EBC3;
   // UNICODE_TO_GBK[14256] := 16#670B;
   // UNICODE_TO_GBK[14257] := 16#C5F3;
   // UNICODE_TO_GBK[14258] := 16#670C;
   // UNICODE_TO_GBK[14259] := 16#9644;
   // UNICODE_TO_GBK[14260] := 16#670D;
   // UNICODE_TO_GBK[14261] := 16#B7FE;
   // UNICODE_TO_GBK[14262] := 16#670E;
   // UNICODE_TO_GBK[14263] := 16#9645;
   // UNICODE_TO_GBK[14264] := 16#670F;
   // UNICODE_TO_GBK[14265] := 16#9646;
   // UNICODE_TO_GBK[14266] := 16#6710;
   // UNICODE_TO_GBK[14267] := 16#EBD4;
   // UNICODE_TO_GBK[14268] := 16#6711;
   // UNICODE_TO_GBK[14269] := 16#9647;
   // UNICODE_TO_GBK[14270] := 16#6712;
   // UNICODE_TO_GBK[14271] := 16#9648;
   // UNICODE_TO_GBK[14272] := 16#6713;
   // UNICODE_TO_GBK[14273] := 16#9649;
   // UNICODE_TO_GBK[14274] := 16#6714;
   // UNICODE_TO_GBK[14275] := 16#CBB7;
   // UNICODE_TO_GBK[14276] := 16#6715;
   // UNICODE_TO_GBK[14277] := 16#EBDE;
   // UNICODE_TO_GBK[14278] := 16#6716;
   // UNICODE_TO_GBK[14279] := 16#964A;
   // UNICODE_TO_GBK[14280] := 16#6717;
   // UNICODE_TO_GBK[14281] := 16#C0CA;
   // UNICODE_TO_GBK[14282] := 16#6718;
   // UNICODE_TO_GBK[14283] := 16#964B;
   // UNICODE_TO_GBK[14284] := 16#6719;
   // UNICODE_TO_GBK[14285] := 16#964C;
   // UNICODE_TO_GBK[14286] := 16#671A;
   // UNICODE_TO_GBK[14287] := 16#964D;
   // UNICODE_TO_GBK[14288] := 16#671B;
   // UNICODE_TO_GBK[14289] := 16#CDFB;
   // UNICODE_TO_GBK[14290] := 16#671C;
   // UNICODE_TO_GBK[14291] := 16#964E;
   // UNICODE_TO_GBK[14292] := 16#671D;
   // UNICODE_TO_GBK[14293] := 16#B3AF;
   // UNICODE_TO_GBK[14294] := 16#671E;
   // UNICODE_TO_GBK[14295] := 16#964F;
   // UNICODE_TO_GBK[14296] := 16#671F;
   // UNICODE_TO_GBK[14297] := 16#C6DA;
   // UNICODE_TO_GBK[14298] := 16#6720;
   // UNICODE_TO_GBK[14299] := 16#9650;
   // UNICODE_TO_GBK[14300] := 16#6721;
   // UNICODE_TO_GBK[14301] := 16#9651;
   // UNICODE_TO_GBK[14302] := 16#6722;
   // UNICODE_TO_GBK[14303] := 16#9652;
   // UNICODE_TO_GBK[14304] := 16#6723;
   // UNICODE_TO_GBK[14305] := 16#9653;
   // UNICODE_TO_GBK[14306] := 16#6724;
   // UNICODE_TO_GBK[14307] := 16#9654;
   // UNICODE_TO_GBK[14308] := 16#6725;
   // UNICODE_TO_GBK[14309] := 16#9655;
   // UNICODE_TO_GBK[14310] := 16#6726;
   // UNICODE_TO_GBK[14311] := 16#EBFC;
   // UNICODE_TO_GBK[14312] := 16#6727;
   // UNICODE_TO_GBK[14313] := 16#9656;
   // UNICODE_TO_GBK[14314] := 16#6728;
   // UNICODE_TO_GBK[14315] := 16#C4BE;
   // UNICODE_TO_GBK[14316] := 16#6729;
   // UNICODE_TO_GBK[14317] := 16#9657;
   // UNICODE_TO_GBK[14318] := 16#672A;
   // UNICODE_TO_GBK[14319] := 16#CEB4;
   // UNICODE_TO_GBK[14320] := 16#672B;
   // UNICODE_TO_GBK[14321] := 16#C4A9;
   // UNICODE_TO_GBK[14322] := 16#672C;
   // UNICODE_TO_GBK[14323] := 16#B1BE;
   // UNICODE_TO_GBK[14324] := 16#672D;
   // UNICODE_TO_GBK[14325] := 16#D4FD;
   // UNICODE_TO_GBK[14326] := 16#672E;
   // UNICODE_TO_GBK[14327] := 16#9658;
   // UNICODE_TO_GBK[14328] := 16#672F;
   // UNICODE_TO_GBK[14329] := 16#CAF5;
   // UNICODE_TO_GBK[14330] := 16#6730;
   // UNICODE_TO_GBK[14331] := 16#9659;
   // UNICODE_TO_GBK[14332] := 16#6731;
   // UNICODE_TO_GBK[14333] := 16#D6EC;
   // UNICODE_TO_GBK[14334] := 16#6732;
   // UNICODE_TO_GBK[14335] := 16#965A;
   // UNICODE_TO_GBK[14336] := 16#6733;
   // UNICODE_TO_GBK[14337] := 16#965B;
   // UNICODE_TO_GBK[14338] := 16#6734;
   // UNICODE_TO_GBK[14339] := 16#C6D3;
   // UNICODE_TO_GBK[14340] := 16#6735;
   // UNICODE_TO_GBK[14341] := 16#B6E4;
   // UNICODE_TO_GBK[14342] := 16#6736;
   // UNICODE_TO_GBK[14343] := 16#965C;
   // UNICODE_TO_GBK[14344] := 16#6737;
   // UNICODE_TO_GBK[14345] := 16#965D;
   // UNICODE_TO_GBK[14346] := 16#6738;
   // UNICODE_TO_GBK[14347] := 16#965E;
   // UNICODE_TO_GBK[14348] := 16#6739;
   // UNICODE_TO_GBK[14349] := 16#965F;
   // UNICODE_TO_GBK[14350] := 16#673A;
   // UNICODE_TO_GBK[14351] := 16#BBFA;
   // UNICODE_TO_GBK[14352] := 16#673B;
   // UNICODE_TO_GBK[14353] := 16#9660;
   // UNICODE_TO_GBK[14354] := 16#673C;
   // UNICODE_TO_GBK[14355] := 16#9661;
   // UNICODE_TO_GBK[14356] := 16#673D;
   // UNICODE_TO_GBK[14357] := 16#D0E0;
   // UNICODE_TO_GBK[14358] := 16#673E;
   // UNICODE_TO_GBK[14359] := 16#9662;
   // UNICODE_TO_GBK[14360] := 16#673F;
   // UNICODE_TO_GBK[14361] := 16#9663;
   // UNICODE_TO_GBK[14362] := 16#6740;
   // UNICODE_TO_GBK[14363] := 16#C9B1;
   // UNICODE_TO_GBK[14364] := 16#6741;
   // UNICODE_TO_GBK[14365] := 16#9664;
   // UNICODE_TO_GBK[14366] := 16#6742;
   // UNICODE_TO_GBK[14367] := 16#D4D3;
   // UNICODE_TO_GBK[14368] := 16#6743;
   // UNICODE_TO_GBK[14369] := 16#C8A8;
   // UNICODE_TO_GBK[14370] := 16#6744;
   // UNICODE_TO_GBK[14371] := 16#9665;
   // UNICODE_TO_GBK[14372] := 16#6745;
   // UNICODE_TO_GBK[14373] := 16#9666;
   // UNICODE_TO_GBK[14374] := 16#6746;
   // UNICODE_TO_GBK[14375] := 16#B8CB;
   // UNICODE_TO_GBK[14376] := 16#6747;
   // UNICODE_TO_GBK[14377] := 16#9667;
   // UNICODE_TO_GBK[14378] := 16#6748;
   // UNICODE_TO_GBK[14379] := 16#E8BE;
   // UNICODE_TO_GBK[14380] := 16#6749;
   // UNICODE_TO_GBK[14381] := 16#C9BC;
   // UNICODE_TO_GBK[14382] := 16#674A;
   // UNICODE_TO_GBK[14383] := 16#9668;
   // UNICODE_TO_GBK[14384] := 16#674B;
   // UNICODE_TO_GBK[14385] := 16#9669;
   // UNICODE_TO_GBK[14386] := 16#674C;
   // UNICODE_TO_GBK[14387] := 16#E8BB;
   // UNICODE_TO_GBK[14388] := 16#674D;
   // UNICODE_TO_GBK[14389] := 16#966A;
   // UNICODE_TO_GBK[14390] := 16#674E;
   // UNICODE_TO_GBK[14391] := 16#C0EE;
   // UNICODE_TO_GBK[14392] := 16#674F;
   // UNICODE_TO_GBK[14393] := 16#D0D3;
   // UNICODE_TO_GBK[14394] := 16#6750;
   // UNICODE_TO_GBK[14395] := 16#B2C4;
   // UNICODE_TO_GBK[14396] := 16#6751;
   // UNICODE_TO_GBK[14397] := 16#B4E5;
   // UNICODE_TO_GBK[14398] := 16#6752;
   // UNICODE_TO_GBK[14399] := 16#966B;
   // UNICODE_TO_GBK[14400] := 16#6753;
   // UNICODE_TO_GBK[14401] := 16#E8BC;
   // UNICODE_TO_GBK[14402] := 16#6754;
   // UNICODE_TO_GBK[14403] := 16#966C;
   // UNICODE_TO_GBK[14404] := 16#6755;
   // UNICODE_TO_GBK[14405] := 16#966D;
   // UNICODE_TO_GBK[14406] := 16#6756;
   // UNICODE_TO_GBK[14407] := 16#D5C8;
   // UNICODE_TO_GBK[14408] := 16#6757;
   // UNICODE_TO_GBK[14409] := 16#966E;
   // UNICODE_TO_GBK[14410] := 16#6758;
   // UNICODE_TO_GBK[14411] := 16#966F;
   // UNICODE_TO_GBK[14412] := 16#6759;
   // UNICODE_TO_GBK[14413] := 16#9670;
   // UNICODE_TO_GBK[14414] := 16#675A;
   // UNICODE_TO_GBK[14415] := 16#9671;
   // UNICODE_TO_GBK[14416] := 16#675B;
   // UNICODE_TO_GBK[14417] := 16#9672;
   // UNICODE_TO_GBK[14418] := 16#675C;
   // UNICODE_TO_GBK[14419] := 16#B6C5;
   // UNICODE_TO_GBK[14420] := 16#675D;
   // UNICODE_TO_GBK[14421] := 16#9673;
   // UNICODE_TO_GBK[14422] := 16#675E;
   // UNICODE_TO_GBK[14423] := 16#E8BD;
   // UNICODE_TO_GBK[14424] := 16#675F;
   // UNICODE_TO_GBK[14425] := 16#CAF8;
   // UNICODE_TO_GBK[14426] := 16#6760;
   // UNICODE_TO_GBK[14427] := 16#B8DC;
   // UNICODE_TO_GBK[14428] := 16#6761;
   // UNICODE_TO_GBK[14429] := 16#CCF5;
   // UNICODE_TO_GBK[14430] := 16#6762;
   // UNICODE_TO_GBK[14431] := 16#9674;
   // UNICODE_TO_GBK[14432] := 16#6763;
   // UNICODE_TO_GBK[14433] := 16#9675;
   // UNICODE_TO_GBK[14434] := 16#6764;
   // UNICODE_TO_GBK[14435] := 16#9676;
   // UNICODE_TO_GBK[14436] := 16#6765;
   // UNICODE_TO_GBK[14437] := 16#C0B4;
   // UNICODE_TO_GBK[14438] := 16#6766;
   // UNICODE_TO_GBK[14439] := 16#9677;
   // UNICODE_TO_GBK[14440] := 16#6767;
   // UNICODE_TO_GBK[14441] := 16#9678;
   // UNICODE_TO_GBK[14442] := 16#6768;
   // UNICODE_TO_GBK[14443] := 16#D1EE;
   // UNICODE_TO_GBK[14444] := 16#6769;
   // UNICODE_TO_GBK[14445] := 16#E8BF;
   // UNICODE_TO_GBK[14446] := 16#676A;
   // UNICODE_TO_GBK[14447] := 16#E8C2;
   // UNICODE_TO_GBK[14448] := 16#676B;
   // UNICODE_TO_GBK[14449] := 16#9679;
   // UNICODE_TO_GBK[14450] := 16#676C;
   // UNICODE_TO_GBK[14451] := 16#967A;
   // UNICODE_TO_GBK[14452] := 16#676D;
   // UNICODE_TO_GBK[14453] := 16#BABC;
   // UNICODE_TO_GBK[14454] := 16#676E;
   // UNICODE_TO_GBK[14455] := 16#967B;
   // UNICODE_TO_GBK[14456] := 16#676F;
   // UNICODE_TO_GBK[14457] := 16#B1AD;
   // UNICODE_TO_GBK[14458] := 16#6770;
   // UNICODE_TO_GBK[14459] := 16#BDDC;
   // UNICODE_TO_GBK[14460] := 16#6771;
   // UNICODE_TO_GBK[14461] := 16#967C;
   // UNICODE_TO_GBK[14462] := 16#6772;
   // UNICODE_TO_GBK[14463] := 16#EABD;
   // UNICODE_TO_GBK[14464] := 16#6773;
   // UNICODE_TO_GBK[14465] := 16#E8C3;
   // UNICODE_TO_GBK[14466] := 16#6774;
   // UNICODE_TO_GBK[14467] := 16#967D;
   // UNICODE_TO_GBK[14468] := 16#6775;
   // UNICODE_TO_GBK[14469] := 16#E8C6;
   // UNICODE_TO_GBK[14470] := 16#6776;
   // UNICODE_TO_GBK[14471] := 16#967E;
   // UNICODE_TO_GBK[14472] := 16#6777;
   // UNICODE_TO_GBK[14473] := 16#E8CB;
   // UNICODE_TO_GBK[14474] := 16#6778;
   // UNICODE_TO_GBK[14475] := 16#9680;
   // UNICODE_TO_GBK[14476] := 16#6779;
   // UNICODE_TO_GBK[14477] := 16#9681;
   // UNICODE_TO_GBK[14478] := 16#677A;
   // UNICODE_TO_GBK[14479] := 16#9682;
   // UNICODE_TO_GBK[14480] := 16#677B;
   // UNICODE_TO_GBK[14481] := 16#9683;
   // UNICODE_TO_GBK[14482] := 16#677C;
   // UNICODE_TO_GBK[14483] := 16#E8CC;
   // UNICODE_TO_GBK[14484] := 16#677D;
   // UNICODE_TO_GBK[14485] := 16#9684;
   // UNICODE_TO_GBK[14486] := 16#677E;
   // UNICODE_TO_GBK[14487] := 16#CBC9;
   // UNICODE_TO_GBK[14488] := 16#677F;
   // UNICODE_TO_GBK[14489] := 16#B0E5;
   // UNICODE_TO_GBK[14490] := 16#6780;
   // UNICODE_TO_GBK[14491] := 16#9685;
   // UNICODE_TO_GBK[14492] := 16#6781;
   // UNICODE_TO_GBK[14493] := 16#BCAB;
   // UNICODE_TO_GBK[14494] := 16#6782;
   // UNICODE_TO_GBK[14495] := 16#9686;
   // UNICODE_TO_GBK[14496] := 16#6783;
   // UNICODE_TO_GBK[14497] := 16#9687;
   // UNICODE_TO_GBK[14498] := 16#6784;
   // UNICODE_TO_GBK[14499] := 16#B9B9;
   // UNICODE_TO_GBK[14500] := 16#6785;
   // UNICODE_TO_GBK[14501] := 16#9688;
   // UNICODE_TO_GBK[14502] := 16#6786;
   // UNICODE_TO_GBK[14503] := 16#9689;
   // UNICODE_TO_GBK[14504] := 16#6787;
   // UNICODE_TO_GBK[14505] := 16#E8C1;
   // UNICODE_TO_GBK[14506] := 16#6788;
   // UNICODE_TO_GBK[14507] := 16#968A;
   // UNICODE_TO_GBK[14508] := 16#6789;
   // UNICODE_TO_GBK[14509] := 16#CDF7;
   // UNICODE_TO_GBK[14510] := 16#678A;
   // UNICODE_TO_GBK[14511] := 16#968B;
   // UNICODE_TO_GBK[14512] := 16#678B;
   // UNICODE_TO_GBK[14513] := 16#E8CA;
   // UNICODE_TO_GBK[14514] := 16#678C;
   // UNICODE_TO_GBK[14515] := 16#968C;
   // UNICODE_TO_GBK[14516] := 16#678D;
   // UNICODE_TO_GBK[14517] := 16#968D;
   // UNICODE_TO_GBK[14518] := 16#678E;
   // UNICODE_TO_GBK[14519] := 16#968E;
   // UNICODE_TO_GBK[14520] := 16#678F;
   // UNICODE_TO_GBK[14521] := 16#968F;
   // UNICODE_TO_GBK[14522] := 16#6790;
   // UNICODE_TO_GBK[14523] := 16#CEF6;
   // UNICODE_TO_GBK[14524] := 16#6791;
   // UNICODE_TO_GBK[14525] := 16#9690;
   // UNICODE_TO_GBK[14526] := 16#6792;
   // UNICODE_TO_GBK[14527] := 16#9691;
   // UNICODE_TO_GBK[14528] := 16#6793;
   // UNICODE_TO_GBK[14529] := 16#9692;
   // UNICODE_TO_GBK[14530] := 16#6794;
   // UNICODE_TO_GBK[14531] := 16#9693;
   // UNICODE_TO_GBK[14532] := 16#6795;
   // UNICODE_TO_GBK[14533] := 16#D5ED;
   // UNICODE_TO_GBK[14534] := 16#6796;
   // UNICODE_TO_GBK[14535] := 16#9694;
   // UNICODE_TO_GBK[14536] := 16#6797;
   // UNICODE_TO_GBK[14537] := 16#C1D6;
   // UNICODE_TO_GBK[14538] := 16#6798;
   // UNICODE_TO_GBK[14539] := 16#E8C4;
   // UNICODE_TO_GBK[14540] := 16#6799;
   // UNICODE_TO_GBK[14541] := 16#9695;
   // UNICODE_TO_GBK[14542] := 16#679A;
   // UNICODE_TO_GBK[14543] := 16#C3B6;
   // UNICODE_TO_GBK[14544] := 16#679B;
   // UNICODE_TO_GBK[14545] := 16#9696;
   // UNICODE_TO_GBK[14546] := 16#679C;
   // UNICODE_TO_GBK[14547] := 16#B9FB;
   // UNICODE_TO_GBK[14548] := 16#679D;
   // UNICODE_TO_GBK[14549] := 16#D6A6;
   // UNICODE_TO_GBK[14550] := 16#679E;
   // UNICODE_TO_GBK[14551] := 16#E8C8;
   // UNICODE_TO_GBK[14552] := 16#679F;
   // UNICODE_TO_GBK[14553] := 16#9697;
   // UNICODE_TO_GBK[14554] := 16#67A0;
   // UNICODE_TO_GBK[14555] := 16#9698;
   // UNICODE_TO_GBK[14556] := 16#67A1;
   // UNICODE_TO_GBK[14557] := 16#9699;
   // UNICODE_TO_GBK[14558] := 16#67A2;
   // UNICODE_TO_GBK[14559] := 16#CAE0;
   // UNICODE_TO_GBK[14560] := 16#67A3;
   // UNICODE_TO_GBK[14561] := 16#D4E6;
   // UNICODE_TO_GBK[14562] := 16#67A4;
   // UNICODE_TO_GBK[14563] := 16#969A;
   // UNICODE_TO_GBK[14564] := 16#67A5;
   // UNICODE_TO_GBK[14565] := 16#E8C0;
   // UNICODE_TO_GBK[14566] := 16#67A6;
   // UNICODE_TO_GBK[14567] := 16#969B;
   // UNICODE_TO_GBK[14568] := 16#67A7;
   // UNICODE_TO_GBK[14569] := 16#E8C5;
   // UNICODE_TO_GBK[14570] := 16#67A8;
   // UNICODE_TO_GBK[14571] := 16#E8C7;
   // UNICODE_TO_GBK[14572] := 16#67A9;
   // UNICODE_TO_GBK[14573] := 16#969C;
   // UNICODE_TO_GBK[14574] := 16#67AA;
   // UNICODE_TO_GBK[14575] := 16#C7B9;
   // UNICODE_TO_GBK[14576] := 16#67AB;
   // UNICODE_TO_GBK[14577] := 16#B7E3;
   // UNICODE_TO_GBK[14578] := 16#67AC;
   // UNICODE_TO_GBK[14579] := 16#969D;
   // UNICODE_TO_GBK[14580] := 16#67AD;
   // UNICODE_TO_GBK[14581] := 16#E8C9;
   // UNICODE_TO_GBK[14582] := 16#67AE;
   // UNICODE_TO_GBK[14583] := 16#969E;
   // UNICODE_TO_GBK[14584] := 16#67AF;
   // UNICODE_TO_GBK[14585] := 16#BFDD;
   // UNICODE_TO_GBK[14586] := 16#67B0;
   // UNICODE_TO_GBK[14587] := 16#E8D2;
   // UNICODE_TO_GBK[14588] := 16#67B1;
   // UNICODE_TO_GBK[14589] := 16#969F;
   // UNICODE_TO_GBK[14590] := 16#67B2;
   // UNICODE_TO_GBK[14591] := 16#96A0;
   // UNICODE_TO_GBK[14592] := 16#67B3;
   // UNICODE_TO_GBK[14593] := 16#E8D7;
   // UNICODE_TO_GBK[14594] := 16#67B4;
   // UNICODE_TO_GBK[14595] := 16#96A1;
   // UNICODE_TO_GBK[14596] := 16#67B5;
   // UNICODE_TO_GBK[14597] := 16#E8D5;
   // UNICODE_TO_GBK[14598] := 16#67B6;
   // UNICODE_TO_GBK[14599] := 16#BCDC;
   // UNICODE_TO_GBK[14600] := 16#67B7;
   // UNICODE_TO_GBK[14601] := 16#BCCF;
   // UNICODE_TO_GBK[14602] := 16#67B8;
   // UNICODE_TO_GBK[14603] := 16#E8DB;
   // UNICODE_TO_GBK[14604] := 16#67B9;
   // UNICODE_TO_GBK[14605] := 16#96A2;
   // UNICODE_TO_GBK[14606] := 16#67BA;
   // UNICODE_TO_GBK[14607] := 16#96A3;
   // UNICODE_TO_GBK[14608] := 16#67BB;
   // UNICODE_TO_GBK[14609] := 16#96A4;
   // UNICODE_TO_GBK[14610] := 16#67BC;
   // UNICODE_TO_GBK[14611] := 16#96A5;
   // UNICODE_TO_GBK[14612] := 16#67BD;
   // UNICODE_TO_GBK[14613] := 16#96A6;
   // UNICODE_TO_GBK[14614] := 16#67BE;
   // UNICODE_TO_GBK[14615] := 16#96A7;
   // UNICODE_TO_GBK[14616] := 16#67BF;
   // UNICODE_TO_GBK[14617] := 16#96A8;
   // UNICODE_TO_GBK[14618] := 16#67C0;
   // UNICODE_TO_GBK[14619] := 16#96A9;
   // UNICODE_TO_GBK[14620] := 16#67C1;
   // UNICODE_TO_GBK[14621] := 16#E8DE;
   // UNICODE_TO_GBK[14622] := 16#67C2;
   // UNICODE_TO_GBK[14623] := 16#96AA;
   // UNICODE_TO_GBK[14624] := 16#67C3;
   // UNICODE_TO_GBK[14625] := 16#E8DA;
   // UNICODE_TO_GBK[14626] := 16#67C4;
   // UNICODE_TO_GBK[14627] := 16#B1FA;
   // UNICODE_TO_GBK[14628] := 16#67C5;
   // UNICODE_TO_GBK[14629] := 16#96AB;
   // UNICODE_TO_GBK[14630] := 16#67C6;
   // UNICODE_TO_GBK[14631] := 16#96AC;
   // UNICODE_TO_GBK[14632] := 16#67C7;
   // UNICODE_TO_GBK[14633] := 16#96AD;
   // UNICODE_TO_GBK[14634] := 16#67C8;
   // UNICODE_TO_GBK[14635] := 16#96AE;
   // UNICODE_TO_GBK[14636] := 16#67C9;
   // UNICODE_TO_GBK[14637] := 16#96AF;
   // UNICODE_TO_GBK[14638] := 16#67CA;
   // UNICODE_TO_GBK[14639] := 16#96B0;
   // UNICODE_TO_GBK[14640] := 16#67CB;
   // UNICODE_TO_GBK[14641] := 16#96B1;
   // UNICODE_TO_GBK[14642] := 16#67CC;
   // UNICODE_TO_GBK[14643] := 16#96B2;
   // UNICODE_TO_GBK[14644] := 16#67CD;
   // UNICODE_TO_GBK[14645] := 16#96B3;
   // UNICODE_TO_GBK[14646] := 16#67CE;
   // UNICODE_TO_GBK[14647] := 16#96B4;
   // UNICODE_TO_GBK[14648] := 16#67CF;
   // UNICODE_TO_GBK[14649] := 16#B0D8;
   // UNICODE_TO_GBK[14650] := 16#67D0;
   // UNICODE_TO_GBK[14651] := 16#C4B3;
   // UNICODE_TO_GBK[14652] := 16#67D1;
   // UNICODE_TO_GBK[14653] := 16#B8CC;
   // UNICODE_TO_GBK[14654] := 16#67D2;
   // UNICODE_TO_GBK[14655] := 16#C6E2;
   // UNICODE_TO_GBK[14656] := 16#67D3;
   // UNICODE_TO_GBK[14657] := 16#C8BE;
   // UNICODE_TO_GBK[14658] := 16#67D4;
   // UNICODE_TO_GBK[14659] := 16#C8E1;
   // UNICODE_TO_GBK[14660] := 16#67D5;
   // UNICODE_TO_GBK[14661] := 16#96B5;
   // UNICODE_TO_GBK[14662] := 16#67D6;
   // UNICODE_TO_GBK[14663] := 16#96B6;
   // UNICODE_TO_GBK[14664] := 16#67D7;
   // UNICODE_TO_GBK[14665] := 16#96B7;
   // UNICODE_TO_GBK[14666] := 16#67D8;
   // UNICODE_TO_GBK[14667] := 16#E8CF;
   // UNICODE_TO_GBK[14668] := 16#67D9;
   // UNICODE_TO_GBK[14669] := 16#E8D4;
   // UNICODE_TO_GBK[14670] := 16#67DA;
   // UNICODE_TO_GBK[14671] := 16#E8D6;
   // UNICODE_TO_GBK[14672] := 16#67DB;
   // UNICODE_TO_GBK[14673] := 16#96B8;
   // UNICODE_TO_GBK[14674] := 16#67DC;
   // UNICODE_TO_GBK[14675] := 16#B9F1;
   // UNICODE_TO_GBK[14676] := 16#67DD;
   // UNICODE_TO_GBK[14677] := 16#E8D8;
   // UNICODE_TO_GBK[14678] := 16#67DE;
   // UNICODE_TO_GBK[14679] := 16#D7F5;
   // UNICODE_TO_GBK[14680] := 16#67DF;
   // UNICODE_TO_GBK[14681] := 16#96B9;
   // UNICODE_TO_GBK[14682] := 16#67E0;
   // UNICODE_TO_GBK[14683] := 16#C4FB;
   // UNICODE_TO_GBK[14684] := 16#67E1;
   // UNICODE_TO_GBK[14685] := 16#96BA;
   // UNICODE_TO_GBK[14686] := 16#67E2;
   // UNICODE_TO_GBK[14687] := 16#E8DC;
   // UNICODE_TO_GBK[14688] := 16#67E3;
   // UNICODE_TO_GBK[14689] := 16#96BB;
   // UNICODE_TO_GBK[14690] := 16#67E4;
   // UNICODE_TO_GBK[14691] := 16#96BC;
   // UNICODE_TO_GBK[14692] := 16#67E5;
   // UNICODE_TO_GBK[14693] := 16#B2E9;
   // UNICODE_TO_GBK[14694] := 16#67E6;
   // UNICODE_TO_GBK[14695] := 16#96BD;
   // UNICODE_TO_GBK[14696] := 16#67E7;
   // UNICODE_TO_GBK[14697] := 16#96BE;
   // UNICODE_TO_GBK[14698] := 16#67E8;
   // UNICODE_TO_GBK[14699] := 16#96BF;
   // UNICODE_TO_GBK[14700] := 16#67E9;
   // UNICODE_TO_GBK[14701] := 16#E8D1;
   // UNICODE_TO_GBK[14702] := 16#67EA;
   // UNICODE_TO_GBK[14703] := 16#96C0;
   // UNICODE_TO_GBK[14704] := 16#67EB;
   // UNICODE_TO_GBK[14705] := 16#96C1;
   // UNICODE_TO_GBK[14706] := 16#67EC;
   // UNICODE_TO_GBK[14707] := 16#BCED;
   // UNICODE_TO_GBK[14708] := 16#67ED;
   // UNICODE_TO_GBK[14709] := 16#96C2;
   // UNICODE_TO_GBK[14710] := 16#67EE;
   // UNICODE_TO_GBK[14711] := 16#96C3;
   // UNICODE_TO_GBK[14712] := 16#67EF;
   // UNICODE_TO_GBK[14713] := 16#BFC2;
   // UNICODE_TO_GBK[14714] := 16#67F0;
   // UNICODE_TO_GBK[14715] := 16#E8CD;
   // UNICODE_TO_GBK[14716] := 16#67F1;
   // UNICODE_TO_GBK[14717] := 16#D6F9;
   // UNICODE_TO_GBK[14718] := 16#67F2;
   // UNICODE_TO_GBK[14719] := 16#96C4;
   // UNICODE_TO_GBK[14720] := 16#67F3;
   // UNICODE_TO_GBK[14721] := 16#C1F8;
   // UNICODE_TO_GBK[14722] := 16#67F4;
   // UNICODE_TO_GBK[14723] := 16#B2F1;
   // UNICODE_TO_GBK[14724] := 16#67F5;
   // UNICODE_TO_GBK[14725] := 16#96C5;
   // UNICODE_TO_GBK[14726] := 16#67F6;
   // UNICODE_TO_GBK[14727] := 16#96C6;
   // UNICODE_TO_GBK[14728] := 16#67F7;
   // UNICODE_TO_GBK[14729] := 16#96C7;
   // UNICODE_TO_GBK[14730] := 16#67F8;
   // UNICODE_TO_GBK[14731] := 16#96C8;
   // UNICODE_TO_GBK[14732] := 16#67F9;
   // UNICODE_TO_GBK[14733] := 16#96C9;
   // UNICODE_TO_GBK[14734] := 16#67FA;
   // UNICODE_TO_GBK[14735] := 16#96CA;
   // UNICODE_TO_GBK[14736] := 16#67FB;
   // UNICODE_TO_GBK[14737] := 16#96CB;
   // UNICODE_TO_GBK[14738] := 16#67FC;
   // UNICODE_TO_GBK[14739] := 16#96CC;
   // UNICODE_TO_GBK[14740] := 16#67FD;
   // UNICODE_TO_GBK[14741] := 16#E8DF;
   // UNICODE_TO_GBK[14742] := 16#67FE;
   // UNICODE_TO_GBK[14743] := 16#96CD;
   // UNICODE_TO_GBK[14744] := 16#67FF;
   // UNICODE_TO_GBK[14745] := 16#CAC1;
   // UNICODE_TO_GBK[14746] := 16#6800;
   // UNICODE_TO_GBK[14747] := 16#E8D9;
   // UNICODE_TO_GBK[14748] := 16#6801;
   // UNICODE_TO_GBK[14749] := 16#96CE;
   // UNICODE_TO_GBK[14750] := 16#6802;
   // UNICODE_TO_GBK[14751] := 16#96CF;
   // UNICODE_TO_GBK[14752] := 16#6803;
   // UNICODE_TO_GBK[14753] := 16#96D0;
   // UNICODE_TO_GBK[14754] := 16#6804;
   // UNICODE_TO_GBK[14755] := 16#96D1;
   // UNICODE_TO_GBK[14756] := 16#6805;
   // UNICODE_TO_GBK[14757] := 16#D5A4;
   // UNICODE_TO_GBK[14758] := 16#6806;
   // UNICODE_TO_GBK[14759] := 16#96D2;
   // UNICODE_TO_GBK[14760] := 16#6807;
   // UNICODE_TO_GBK[14761] := 16#B1EA;
   // UNICODE_TO_GBK[14762] := 16#6808;
   // UNICODE_TO_GBK[14763] := 16#D5BB;
   // UNICODE_TO_GBK[14764] := 16#6809;
   // UNICODE_TO_GBK[14765] := 16#E8CE;
   // UNICODE_TO_GBK[14766] := 16#680A;
   // UNICODE_TO_GBK[14767] := 16#E8D0;
   // UNICODE_TO_GBK[14768] := 16#680B;
   // UNICODE_TO_GBK[14769] := 16#B6B0;
   // UNICODE_TO_GBK[14770] := 16#680C;
   // UNICODE_TO_GBK[14771] := 16#E8D3;
   // UNICODE_TO_GBK[14772] := 16#680D;
   // UNICODE_TO_GBK[14773] := 16#96D3;
   // UNICODE_TO_GBK[14774] := 16#680E;
   // UNICODE_TO_GBK[14775] := 16#E8DD;
   // UNICODE_TO_GBK[14776] := 16#680F;
   // UNICODE_TO_GBK[14777] := 16#C0B8;
   // UNICODE_TO_GBK[14778] := 16#6810;
   // UNICODE_TO_GBK[14779] := 16#96D4;
   // UNICODE_TO_GBK[14780] := 16#6811;
   // UNICODE_TO_GBK[14781] := 16#CAF7;
   // UNICODE_TO_GBK[14782] := 16#6812;
   // UNICODE_TO_GBK[14783] := 16#96D5;
   // UNICODE_TO_GBK[14784] := 16#6813;
   // UNICODE_TO_GBK[14785] := 16#CBA8;
   // UNICODE_TO_GBK[14786] := 16#6814;
   // UNICODE_TO_GBK[14787] := 16#96D6;
   // UNICODE_TO_GBK[14788] := 16#6815;
   // UNICODE_TO_GBK[14789] := 16#96D7;
   // UNICODE_TO_GBK[14790] := 16#6816;
   // UNICODE_TO_GBK[14791] := 16#C6DC;
   // UNICODE_TO_GBK[14792] := 16#6817;
   // UNICODE_TO_GBK[14793] := 16#C0F5;
   // UNICODE_TO_GBK[14794] := 16#6818;
   // UNICODE_TO_GBK[14795] := 16#96D8;
   // UNICODE_TO_GBK[14796] := 16#6819;
   // UNICODE_TO_GBK[14797] := 16#96D9;
   // UNICODE_TO_GBK[14798] := 16#681A;
   // UNICODE_TO_GBK[14799] := 16#96DA;
   // UNICODE_TO_GBK[14800] := 16#681B;
   // UNICODE_TO_GBK[14801] := 16#96DB;
   // UNICODE_TO_GBK[14802] := 16#681C;
   // UNICODE_TO_GBK[14803] := 16#96DC;
   // UNICODE_TO_GBK[14804] := 16#681D;
   // UNICODE_TO_GBK[14805] := 16#E8E9;
   // UNICODE_TO_GBK[14806] := 16#681E;
   // UNICODE_TO_GBK[14807] := 16#96DD;
   // UNICODE_TO_GBK[14808] := 16#681F;
   // UNICODE_TO_GBK[14809] := 16#96DE;
   // UNICODE_TO_GBK[14810] := 16#6820;
   // UNICODE_TO_GBK[14811] := 16#96DF;
   // UNICODE_TO_GBK[14812] := 16#6821;
   // UNICODE_TO_GBK[14813] := 16#D0A3;
   // UNICODE_TO_GBK[14814] := 16#6822;
   // UNICODE_TO_GBK[14815] := 16#96E0;
   // UNICODE_TO_GBK[14816] := 16#6823;
   // UNICODE_TO_GBK[14817] := 16#96E1;
   // UNICODE_TO_GBK[14818] := 16#6824;
   // UNICODE_TO_GBK[14819] := 16#96E2;
   // UNICODE_TO_GBK[14820] := 16#6825;
   // UNICODE_TO_GBK[14821] := 16#96E3;
   // UNICODE_TO_GBK[14822] := 16#6826;
   // UNICODE_TO_GBK[14823] := 16#96E4;
   // UNICODE_TO_GBK[14824] := 16#6827;
   // UNICODE_TO_GBK[14825] := 16#96E5;
